	FUNCTION FC 833  : VOID
	TITLE =MAL1S033 Section control: LINE 1 SEC 33 KILN 2
	//COPYRIGHT:    (C) 2009 BY  BUHLER AG
	//                           CH-9240 UZWIL  SWITZERLAND
	//
	//PRODUCT:      WinCoS_BIW01_09
	//
	//TITLE:        LINE 1 SEC 33 KILN 2
	//                 Section control
	//
	//--------------------------------------------------------------------------------
	//
	//IDENT:        AUTHOR:             DEPT:                              DATE:
	//
	//P01_FC833.1.0 K.Renz              CSB41                              20.Okt.2009
	//              1st Release
	//
	//--------------------------------------------------------------------------------
	//
	//PURPOSE:
	//
	//REFERENCES : GCSOSMAN
	//
	//--------------------------------------------------------------------------------
	//
	//
	AUTHOR  : KR
	FAMILY  : USW
	VERSION : 9.9
	//0000 to 0999: Main Functions
	//              0 =Main Function Cylic
	//              1 =Main Function Coldstart/Newstart
	//              2 =Main Function Warm Start

	VAR_INPUT
	  InCode : INT ;
	END_VAR

	VAR_TEMP
	tmpStartNext : BOOL ;	//Condition to Start next element
	tmpFlagFault : BOOL ;	//Flag mechanical fault
	tmpEnableFeed : BOOL ;
	tmpStartScale : BOOL ;
	tmpStartLiqScale : BOOL ; //Enable to Start Lipquid Scale
	tmpSndBin: Int ;
	tmpRcvBin: Int ;
	tmpBool : BOOL ;
	tmpByte : BYTE ;
	tmpWord : WORD ;
	tmpDWord : DWORD ;
	tmpInt : INT ;
	tmpRET : INT ;
	tmpDInt : DINT ;
	tmpCyclusTime : DINT ;
	tmpWetSteep : BOOL ;
	END_VAR

	BEGIN

	NETWORK
	TITLE =
	//=================================================
	//=================================================
	//S T A R T   M A I N   F U N C T I O N
	//=================================================
	//=================================================
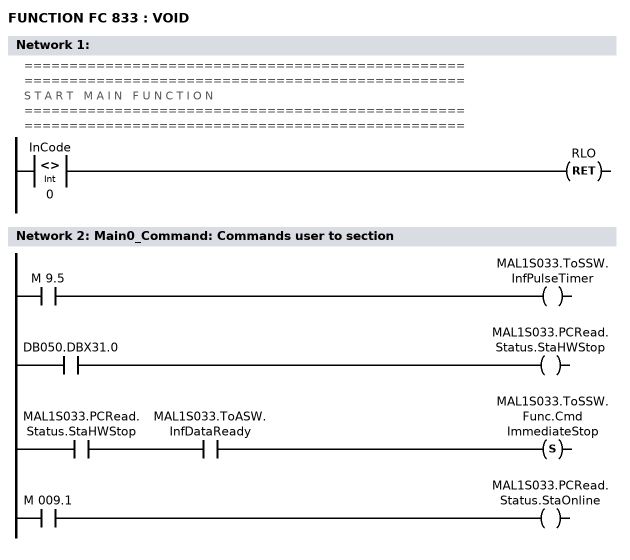
	      L InCode;
	      L 0;
	      <>I;
	      BEB;

	NETWORK
	TITLE =Main0_Command: Commands user to section
	      NOP   0;
	//-Tick 1 second---
		U     M 9.5;
		=     MAL1S033.ToSSW.InfPulseTimer;
	//-Hardware stop---
		U     DB050.DBX31.0 ;
		=     MAL1S033.PCRead.Status.StaHWStop;
		U   MAL1S033.PCRead.Status.StaHWStop;
		U   MAL1S033.ToASW.InfDataReady;
		S     MAL1S033.ToSSW.Func.CmdImmediateStop;
	//-Online---
		U     M 009.1 ;
		=     MAL1S033.PCRead.Status.StaOnline;
	NETWORK
	TITLE =ASW_UC: User commands to section
	NOP 0;
	//-Additional user commands---
	//-GP standard commands---
	      AUF   "MAL1S033" ;
	      L     L#0 ;                           // Enter the differenz of the target weight and prestop weight
	      T    "MAL1S033".VarTemp.InOutValue3;  // Prestop weight
	      CALL FC   120 (
	           InCode                   := 2001);// Section function: Standard section commands

	//-Condition CmdSequenzStop---
	      U     MAL1S033.ToSSW.Func.CmdSequenzStop;
	//      S     "MAL1S033".ToSSW.Func.CmdSequenzStop
	      R     MAL1S033.ToSSW.Func.CmdSequenzStop;
	//-Extended section commands---
	      AUF   "MAL1S033";
	      CALL "STD_LineSecStdSub" (
	           InCode                   := 2002);// Section function: Extended section commands
	//-Status from pulse commands---
	      CLR;
	      =     DB833.DBX  157.0;
	      =     DB833.DBX  157.1;
	      =     DB833.DBX  157.2;
	      =     DB833.DBX  157.3;
	      =     DB833.DBX  157.4;
	      =     DB833.DBX  157.5;
	      =     DB833.DBX  157.6;
	      =     DB833.DBX  157.7;
	//
	NETWORK
	TITLE =Main0_Dest: Destination
	NETWORK
	TITLE =Main0_Next: Ready for next batch

		ON    MAL1S033.ToASW.InfDataReady;
		=     MAL1S033.ToSSW.InfReadyForNewBatch;
	NETWORK
	TITLE =Main0_Control: Control section
	      NOP   0;
	//-Process commands from PCS---
		AUF   "MAL1S033" ;
		CALL FC    60 (// Methode O_Section
		CODE                     := 7);
	//-Process commands from user---
		AUF   "MAL1S033" ;
		CALL FC    60 (// Methode Control
		CODE                     := 0);
	//-Process section step---
		AUF   "MAL1S033" ;
		CALL FC    60 (// Methode Step_execute
		CODE                     := 2);
		AUF   "MAL1S033" ;
		CALL FC    60 (// Methode Step_transition
		CODE                     := 3);
	//-Process section state---
		AUF   "MAL1S033" ;
		CALL FC    60 (// Methode State
		CODE                     := 4);

	NETWORK
	TITLE =Main0_Init: Init
		UN    MAL1S033.ToASW.Transition.ToWait;
		UN    MAL1S033.ToASW.CmdNewBatch;
		SPB   in00;
	//-User initialization---
		AUF   "MAL1S033" ;
	//
	//-Section function: Init ---
		AUF   "MAL1S033" ;
	      CALL FC   120 (
	           InCode                   := 2003);// Section function: Init
	//
	//-Group interface---
	//
	//-Initialise bin objects---
	//
	//-Emptying job---
	      U    MAL1S033.JobAc.StaBatch.StaEmptyingBatch;
	      S     MAL1S033.PCRead.Status.StaLoaded;
	//
	//-Error Batch---
	//
	in00:	NOP   0;

	NETWORK
	TITLE =ASW_VB: Various functions before bin control
	      NOP   0;
	//
	//-Update staSameSndRcv in sender binlist---
	NETWORK
	TITLE =Main0_GrNRS: Not Relevant for started / Fault
		NOP 0;
	NETWORK
	TITLE =Main0_GrSelection: Group selection
	// List of the used objects in the section
	// ==========================
	// G022G       GENERAL ELEMENTS KILN 2
	// G261M       BELT CONVEYOR 7200 KILN
	// G262M       BELT CONVEYOR 7300 KILN
	// G263M       BELT CONVEYOR 7301 KILN
	// G264M       BELT CONVEYOR 7400 KILN
	// G291M       LIFTING DEVICE KILN 2
	// G292M       TRAVELLING DRIVE KILN 2
	// G293M       UNLOADING / LOADING SCREW KILN 2
	// G294M       DISCHARGE DOOR KILN 2
	// G295M       TEMPERATURE MES. KILN 2
	// G296M       AIR SHUT SLIDE KILN 2
	// G297M       FAN KILN 2
	// G298M       FRESH AIR LOUVER KILN 2
	// G299M       RECYCLING AIR FLAP KILN 2
	// G300M       EXHAUST AIR FLAP KILN 2
	// G301M       LOUVER HEATING GLASS TUBE HEAT EXCHANGER
	// G302M       HEATING KILN 2
	// G303M       LOUVER AIR HEATER KILN 2
	// G304M       WITHERING AIR KILN 2
	// G279M       HEATING KILN 1 + 2
	// G305M       CHAIN CONVEYOR 9002 KILN 2
	// G281M       ELEVATOR 9002 AFTER KILN
	// G282M       FLAP BOX 9008
	// G283M       CULM BATCH BIN 9005
	//
	      NOP   0;
//-Condition for preselection---
		U     MAL1S033.ToASW.InfDataReady;
		SPB   GS01;
//-Deselect groups ---
		CALL FB     9 , "GCS7_GrCtrlDBTmp" (// GrCtr.Methode Deselect
		     Code  := 3,
		     Sec   := "MAL1S033".Gr);
		SPA   GS02;
//-Select groups ---
	GS01:	NOP 0;
	//-Prepare for preselection ---
		CALL FB     9 , "GCS7_GrCtrlDBTmp" (// GrCtr.Methode Init Preselection
		     Code  := 1,
		     Sec   := "MAL1S033".Gr);
	//
	//
	//-Prestart used groups --
		U     M     50.0;
		=     M     50.0;

	//-Preselect used groups --
		U     M     50.0;
		=     M     50.0;
		S   MAL1S033.Gr.InPreselect[22];   //-->G022G GENERAL ELEMENTS KILN 2
		S   MAL1S033.Gr.InPreselect[261];   //-->G261M BELT CONVEYOR 7200 KILN
		S   MAL1S033.Gr.InPreselect[262];   //-->G262M BELT CONVEYOR 7300 KILN
		S   MAL1S033.Gr.InPreselect[263];   //-->G263M BELT CONVEYOR 7301 KILN
		S   MAL1S033.Gr.InPreselect[264];   //-->G264M BELT CONVEYOR 7400 KILN
		S   MAL1S033.Gr.InPreselect[291];   //-->G291M LIFTING DEVICE KILN 2
		S   MAL1S033.Gr.InPreselect[292];   //-->G292M TRAVELLING DRIVE KILN 2
		S   MAL1S033.Gr.InPreselect[293];   //-->G293M UNLOADING / LOADING SCREW KILN 2
		S   MAL1S033.Gr.InPreselect[294];   //-->G294M DISCHARGE DOOR KILN 2
		S   MAL1S033.Gr.InPreselect[295];   //-->G295M TEMPERATURE MES. KILN 2
		S   MAL1S033.Gr.InPreselect[296];   //-->G296M AIR SHUT SLIDE KILN 2
		S   MAL1S033.Gr.InPreselect[297];   //-->G297M FAN KILN 2
		S   MAL1S033.Gr.InPreselect[298];   //-->G298M FRESH AIR LOUVER KILN 2
		S   MAL1S033.Gr.InPreselect[299];   //-->G299M RECYCLING AIR FLAP KILN 2
		S   MAL1S033.Gr.InPreselect[300];   //-->G300M EXHAUST AIR FLAP KILN 2
		S   MAL1S033.Gr.InPreselect[301];   //-->G301M LOUVER HEATING GLASS TUBE HEAT EXCHANGER
		S   MAL1S033.Gr.InPreselect[302];   //-->G302M HEATING KILN 2
		S   MAL1S033.Gr.InPreselect[303];   //-->G303M LOUVER AIR HEATER KILN 2
		S   MAL1S033.Gr.InPreselect[304];   //-->G304M WITHERING AIR KILN 2
		S   MAL1S033.Gr.InPreselect[279];   //-->G279M HEATING KILN 1 + 2
		S   MAL1S033.Gr.InPreselect[305];   //-->G305M CHAIN CONVEYOR 9002 KILN 2
		S   MAL1S033.Gr.InPreselect[281];   //-->G281M ELEVATOR 9002 AFTER KILN
		S   MAL1S033.Gr.InPreselect[282];   //-->G282M FLAP BOX 9008
		S   MAL1S033.Gr.InPreselect[283];   //-->G283M CULM BATCH BIN 9005
	      L     1;
	      L     "MAL1S033Par".StepAct.StepNumber;
	      UW;
	      ==I;  // step wetsteep
	      =    "MAL1S033Par".Par.FlagGen.WetStep;

	//
	//-Set CmdNewJob ---
	     U     MAL1S033.Gr.InPreselect[261];
	     UN    #GCS7_GrCtrlDB.OutOccupied[261];
	     S       G261M.CmdNewJob;
	     U     MAL1S033.Gr.InPreselect[262];
	     UN    #GCS7_GrCtrlDB.OutOccupied[262];
	     S       G262M.CmdNewJob;
	     U     MAL1S033.Gr.InPreselect[263];
	     UN    #GCS7_GrCtrlDB.OutOccupied[263];
	     S       G263M.CmdNewJob;
	     U     MAL1S033.Gr.InPreselect[264];
	     UN    #GCS7_GrCtrlDB.OutOccupied[264];
	     S       G264M.CmdNewJob;
	     U     MAL1S033.Gr.InPreselect[291];
	     UN    #GCS7_GrCtrlDB.OutOccupied[291];
	     S       G291M.CmdNewJob;
	     U     MAL1S033.Gr.InPreselect[292];
	     UN    #GCS7_GrCtrlDB.OutOccupied[292];
	     S       G292M.CmdNewJob;
	     U     MAL1S033.Gr.InPreselect[293];
	     UN    #GCS7_GrCtrlDB.OutOccupied[293];
	     S       G293M.CmdNewJob;
	     U     MAL1S033.Gr.InPreselect[294];
	     UN    #GCS7_GrCtrlDB.OutOccupied[294];
	     S       G294M.CmdNewJob;
	     U     MAL1S033.Gr.InPreselect[295];
	     UN    #GCS7_GrCtrlDB.OutOccupied[295];
	     S       G295M.CmdNewJob;
	     U     MAL1S033.Gr.InPreselect[296];
	     UN    #GCS7_GrCtrlDB.OutOccupied[296];
	     S       G296M.CmdNewJob;
	     U     MAL1S033.Gr.InPreselect[297];
	     UN    #GCS7_GrCtrlDB.OutOccupied[297];
	     S       G297M.CmdNewJob;
	     U     MAL1S033.Gr.InPreselect[298];
	     UN    #GCS7_GrCtrlDB.OutOccupied[298];
	     S       G298M.CmdNewJob;
	     U     MAL1S033.Gr.InPreselect[299];
	     UN    #GCS7_GrCtrlDB.OutOccupied[299];
	     S       G299M.CmdNewJob;
	     U     MAL1S033.Gr.InPreselect[300];
	     UN    #GCS7_GrCtrlDB.OutOccupied[300];
	     S       G300M.CmdNewJob;
	     U     MAL1S033.Gr.InPreselect[301];
	     UN    #GCS7_GrCtrlDB.OutOccupied[301];
	     S       G301M.CmdNewJob;
	     U     MAL1S033.Gr.InPreselect[302];
	     UN    #GCS7_GrCtrlDB.OutOccupied[302];
	     S       G302M.CmdNewJob;
	     U     MAL1S033.Gr.InPreselect[303];
	     UN    #GCS7_GrCtrlDB.OutOccupied[303];
	     S       G303M.CmdNewJob;
	     U     MAL1S033.Gr.InPreselect[304];
	     UN    #GCS7_GrCtrlDB.OutOccupied[304];
	     S       G304M.CmdNewJob;
	     U     MAL1S033.Gr.InPreselect[279];
	     UN    #GCS7_GrCtrlDB.OutOccupied[279];
	     S       G279M.CmdNewJob;
	     U     MAL1S033.Gr.InPreselect[305];
	     UN    #GCS7_GrCtrlDB.OutOccupied[305];
	     S       G305M.CmdNewJob;
	     U     MAL1S033.Gr.InPreselect[281];
	     UN    #GCS7_GrCtrlDB.OutOccupied[281];
	     S       G281M.CmdNewJob;
	     U     MAL1S033.Gr.InPreselect[282];
	     UN    #GCS7_GrCtrlDB.OutOccupied[282];
	     S       G282M.CmdNewJob;
	     U     MAL1S033.Gr.InPreselect[283];
	     UN    #GCS7_GrCtrlDB.OutOccupied[283];
	     S       G283M.CmdNewJob;
	//
	//
	//-Test preselected groups ---
		CALL FB     9 , "GCS7_GrCtrlDBTmp" (// GrCtr.Methode Select
		     Code  := 2,
		     Sec   := "MAL1S033".Gr);
	//
	//-Way conflict if not available---
		CLR;
		S     MAL1S033.Gr.All.OutGrConflict;
	//
	//-Test occupied real and virtual groups---
	GS02:   NOP 0;
		U     MAL1S033.Gr.All.OutSelectionValid;
		UN    MAL1S033.Gr.All.OutGrIsLocked;
		=     MAL1S033.Gr.All.InOutASWSelectionOK;
	//
	//
	//----- Send data to selected groups =====
	GS3:	UN  MAL1S033.Gr.OutSelected[261]; //G261M
		SPB GS4;
		L     "MAL1".Para.ParLineNr;
		T     G261M.Gr.InLine;
	GS4:	UN  MAL1S033.Gr.OutSelected[262]; //G262M
		SPB GS5;
		L     "MAL1".Para.ParLineNr;
		T     G262M.Gr.InLine;
	GS5:	UN  MAL1S033.Gr.OutSelected[263]; //G263M
		SPB GS6;
		L     "MAL1".Para.ParLineNr;
		T     G263M.Gr.InLine;
	GS6:	UN  MAL1S033.Gr.OutSelected[264]; //G264M
		SPB GS7;
		L     "MAL1".Para.ParLineNr;
		T     G264M.Gr.InLine;
	GS7:	UN  MAL1S033.Gr.OutSelected[291]; //G291M
		SPB GS8;
		L     "MAL1".Para.ParLineNr;
		T     G291M.Gr.InLine;
	GS8:	UN  MAL1S033.Gr.OutSelected[292]; //G292M
		SPB GS9;
		L     "MAL1".Para.ParLineNr;
		T     G292M.Gr.InLine;
	GS9:	UN  MAL1S033.Gr.OutSelected[293]; //G293M
		SPB GS10;
		L     "MAL1".Para.ParLineNr;
		T     G293M.Gr.InLine;
	GS10:	UN  MAL1S033.Gr.OutSelected[294]; //G294M
		SPB GS11;
		L     "MAL1".Para.ParLineNr;
		T     G294M.Gr.InLine;
	GS11:	UN  MAL1S033.Gr.OutSelected[295]; //G295M
		SPB GS12;
		L     "MAL1".Para.ParLineNr;
		T     G295M.Gr.InLine;
	GS12:	UN  MAL1S033.Gr.OutSelected[296]; //G296M
		SPB GS13;
		L     "MAL1".Para.ParLineNr;
		T     G296M.Gr.InLine;
	GS13:	UN  MAL1S033.Gr.OutSelected[297]; //G297M
		SPB GS14;
		L     "MAL1".Para.ParLineNr;
		T     G297M.Gr.InLine;
	GS14:	UN  MAL1S033.Gr.OutSelected[298]; //G298M
		SPB GS15;
		L     "MAL1".Para.ParLineNr;
		T     G298M.Gr.InLine;
	GS15:	UN  MAL1S033.Gr.OutSelected[299]; //G299M
		SPB GS16;
		L     "MAL1".Para.ParLineNr;
		T     G299M.Gr.InLine;
	GS16:	UN  MAL1S033.Gr.OutSelected[300]; //G300M
		SPB GS17;
		L     "MAL1".Para.ParLineNr;
		T     G300M.Gr.InLine;
	GS17:	UN  MAL1S033.Gr.OutSelected[301]; //G301M
		SPB GS18;
		L     "MAL1".Para.ParLineNr;
		T     G301M.Gr.InLine;
	GS18:	UN  MAL1S033.Gr.OutSelected[302]; //G302M
		SPB GS19;
		L     "MAL1".Para.ParLineNr;
		T     G302M.Gr.InLine;
	GS19:	UN  MAL1S033.Gr.OutSelected[303]; //G303M
		SPB GS20;
		L     "MAL1".Para.ParLineNr;
		T     G303M.Gr.InLine;
	GS20:	UN  MAL1S033.Gr.OutSelected[304]; //G304M
		SPB GS21;
		L     "MAL1".Para.ParLineNr;
		T     G304M.Gr.InLine;
	GS21:	UN  MAL1S033.Gr.OutSelected[279]; //G279M
		SPB GS22;
		L     "MAL1".Para.ParLineNr;
		T     G279M.Gr.InLine;
	GS22:	UN  MAL1S033.Gr.OutSelected[305]; //G305M
		SPB GS23;
		L     "MAL1".Para.ParLineNr;
		T     G305M.Gr.InLine;
	GS23:	UN  MAL1S033.Gr.OutSelected[281]; //G281M
		SPB GS24;
		L     "MAL1".Para.ParLineNr;
		T     G281M.Gr.InLine;
	GS24:	UN  MAL1S033.Gr.OutSelected[282]; //G282M
		SPB GS25;
		L     "MAL1".Para.ParLineNr;
		T     G282M.Gr.InLine;
	GS25:	UN  MAL1S033.Gr.OutSelected[283]; //G283M
		SPB GS26;
		L     "MAL1".Para.ParLineNr;
		T     G283M.Gr.InLine;
	GS26:	NOP 0;
	NETWORK
	TITLE =Main0_GrCmd: CMD section to Groups

		NOP   0;
//-Way Adjust Time---
		O     MAL1S033.Gr.All.CmdNewSelection;
		O     MAL1S033.ToASW.CmdModify;
		S     MAL1S033.ToSSW.CmdNewWay;
		AUF   "MAL1S033" ;
		CALL FC    60 (// Methode Adjust Time
		CODE                     := 13);
//-Continue---
		U     MAL1S033.ToASW.Func.CmdStart;
		O     MAL1S033.ToASW.Func.CmdNextStep;
		S     MAL1S033.Gr.All.CmdContinue;
//-Fault reset---
		U     MAL1S033.ToASW.Func.CmdFaultReset;
		S     MAL1S033.Gr.All.CmdFaultReset;
//-Manual mode---
		U     MAL1S033.ToASW.Func.CmdAutomatic;
		S     MAL1S033.Gr.All.CmdManualOff;
		UN     MAL1S033.PCRead.Status.StaHand;
		S     MAL1S033.Gr.All.CmdManualOffRel;
//-Clear idling---
		U     MAL1S033.PCRead.Status.StaImmediateStopASW;
		S     MAL1S033.Gr.All.CmdClearIdling;
//-Start next---
		UN    MAL1S033.PCRead.Status.StaStep;
		O     MAL1S033.ToASW.Func.CmdNextStep;
		U(;
		L       MAL1S033.PCRead.OutWayAdjustTime;
		L     2;
		>I;
		O     MAL1S033.ToASW.InfWayAdjustTimeEnd;
		);
		UN    MAL1S033.Gr.All.CmdNewSelection;
		UN    MAL1S033.PCRead.Step.StWait;
		=     #tmpStartNext; //-->VarStartNext
//-Start next feed---
		U     MAL1S033.Gr.Wgr.OutStartedRel;
		ON    MAL1S033.ToASW.InfWayAdjustTimeEnd;
		UN    MAL1S033.PCRead.Status.StaFeedOffASW;
		UN    MAL1S033.PCRead.Status.StaImmediateStopASW;
		U     MAL1S033.Gr.Mgr.OutStartedRel;
		U     MAL1S033.PCRead.Step.StActive;
		=     MAL1S033.Gr.Feed.InEnable;
		=     #tmpEnableFeed;
		U     #tmpStartNext;
		U     MAL1S033.Gr.Wgr.OutStartedRel;
		U     MAL1S033.Gr.All.OutAutoStartOk;
		U     MAL1S033.PCRead.Status.StaAutostartSec;
		=     MAL1S033.Gr.Feed.CmdNext;
//-Start next machine group---
		UN    MAL1S033.PCRead.Status.StaImmediateStopASW;
		=     MAL1S033.Gr.Mgr.InEnable;
		U     #tmpStartNext;
		=     MAL1S033.Gr.Mgr.CmdNext;
//-Start next way group---
		UN    MAL1S033.PCRead.Status.StaImmediateStopASW;
		=     MAL1S033.Gr.Wgr.InEnable;
		UN    MAL1S033.PCRead.Status.StaStep;
		O     MAL1S033.ToASW.Func.CmdNextStep;
		=     MAL1S033.Gr.Wgr.CmdNext;
//-Start next general group---
		UN    MAL1S033.PCRead.Status.StaImmediateStopASW;
		=     MAL1S033.Gr.Ggr.InEnable;
		U     #tmpStartNext;
		=     MAL1S033.Gr.Ggr.CmdNext;
//-Update command state---
		CALL FB     9 , "GCS7_GrCtrlDBTmp" (// GrCtr.Methode UpdateCmdSt
		     Code  := 4,
		     Sec   := "MAL1S033".Gr);

	NETWORK
	TITLE =Main0_Status: Fault/Status

		NOP   0;
//- Autostart Section---
		UN    MAL1S033.ToASW.Func.CmdStart;
		O     MAL1S033.Gr.All.OutAutoStartOk;
		=     MAL1S033.TimeoutAutostart.EN;
		CALL FC18 (
		   IN                       := MAL1S033.TimeoutAutostart.EN,
		   PT                       := 10,
		   Q                        := MAL1S033.TimeoutAutostart.Q,
		ET                       := MAL1S033.TimeoutAutostart.ET);
		U     MAL1S033.TimeoutAutostart.Q;
		UN     MAL1S033.Gr.All.OutAutoStartOk;
		R     MAL1S033.PCRead.Status.StaAutostartSec;
		U     MAL1S033.ToASW.Func.CmdStart;
		ON    MAL1S033.ToASW.InfDataReady;
		S     MAL1S033.PCRead.Status.StaAutostartSec;
//-Stopped---
		UN    MAL1S033.Gr.Mgr.InEnable;
		U     MAL1S033.Gr.All.OutStoppedRel;
		O     MAL1S033.Gr.All.OutStoppedAll;
		UN    MAL1S033.PCRead.Status.StaStep;
		O;
		U     MAL1S033.Gr.Mgr.OutStoppedRel;
		U     MAL1S033.PCRead.Status.StaStep;
		=     MAL1S033.ToSSW.InfStopped;
//-Started---
		U     MAL1S033.Gr.Mgr.OutStartedRel;
		=     MAL1S033.ToSSW.InfStarted;
//-Feeding---
		U     MAL1S033.Gr.Feed.InEnable; //Section without Feed groups
		ON    MAL1S033.Gr.Feed.OutStoppedAll;
		U     MAL1S033.Gr.Feed.OutStartedRel;
		=     MAL1S033.ToSSW.InfFeeding;
//-Autostart---
		U     MAL1S033.Gr.All.OutAutostartOkAll;
		U     MAL1S033.PCRead.Status.StaAutostartSec;
		=     MAL1S033.PCRead.Status.StaAutostart;
//-DPFault---
		U     MAL1S033.Gr.All.OutDPFault;
		=     MAL1S033.PCRead.Status.StaDPFault;
		S       MAL1S033.ToSSW.Func.CmdFeedOff;
//-Startwarning---
		U     MAL1S033.Gr.All.OutStartWarning;
		=     MAL1S033.PCRead.Status.StaStartwarning;
//-Way conflict---
		U     MAL1S033.Gr.All.OutGrConflict;
		=     MAL1S033.PCRead.Fault.EsWayConflict;
//-Warning---
		U     MAL1S033.Gr.All.OutWarning;
		=     MAL1S033.PCRead.Fault.EsWarning;
//-Fault---
		U     MAL1S033.Gr.All.OutFaultRel;
		FP      MAL1S033.PCRead.Fault.EsMech;
		S       MAL1S033.ToSSW.Func.CmdFeedOff;
//-Sender empty---
		CLR;
		=     MAL1S033.PCRead.Fault.EsEmpty; //-->Sec.EsEmpty
//-Receiver full---
		CLR;
		=     MAL1S033.PCRead.Fault.EsFull;

	NETWORK
	TITLE =Main0_StatusASW: Status from ASW
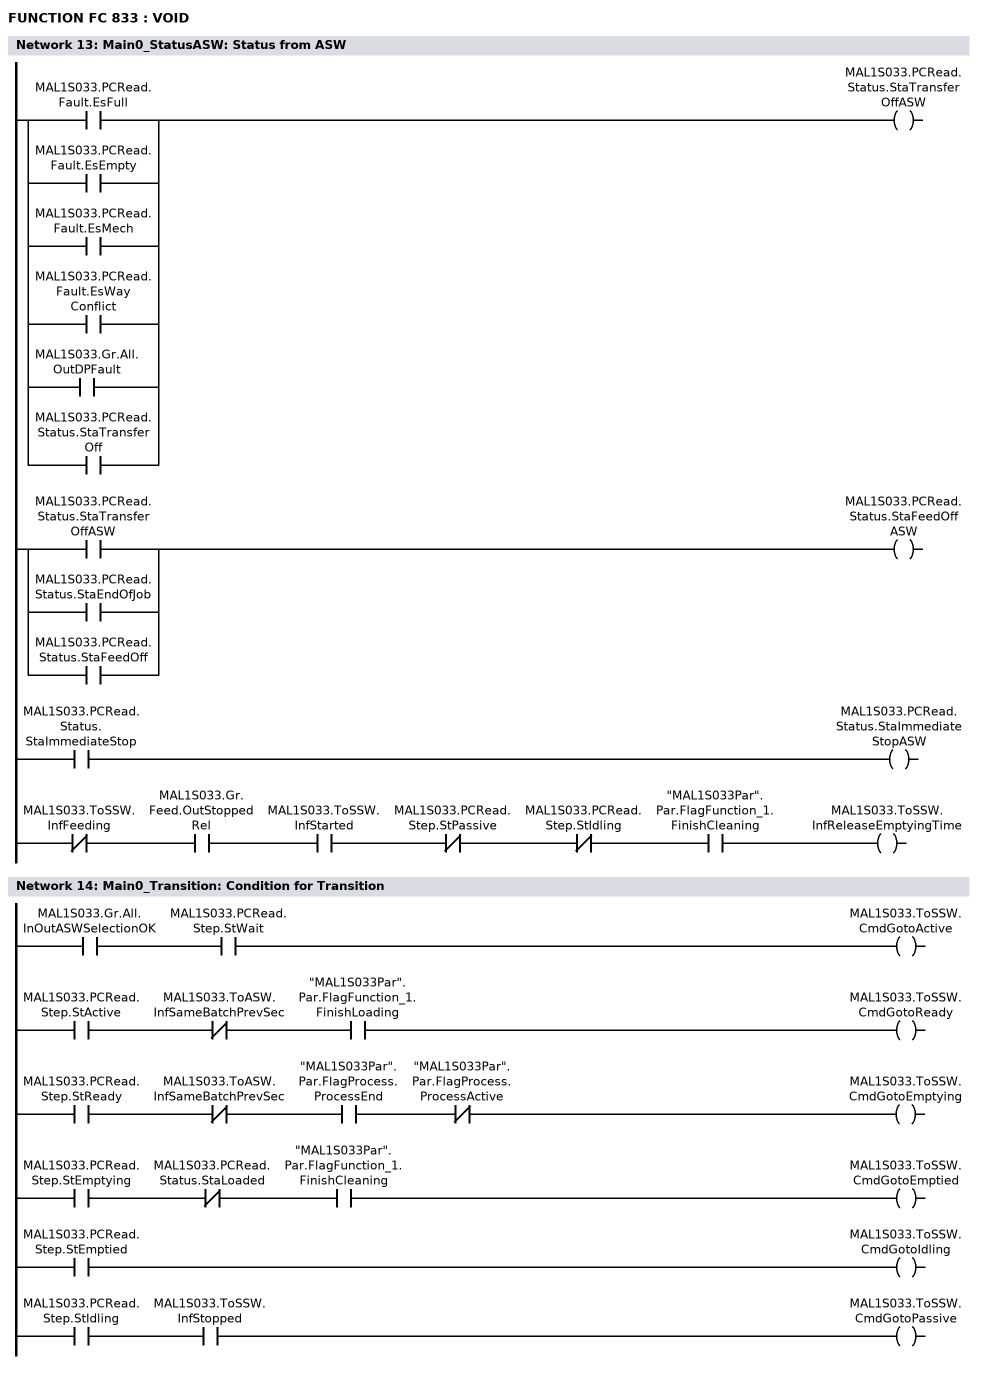
		NOP   0;
//-Transfer off with automatic restart---
		O     MAL1S033.PCRead.Fault.EsFull;
		O     MAL1S033.PCRead.Fault.EsEmpty;
		O     MAL1S033.PCRead.Fault.EsMech;
		O     MAL1S033.PCRead.Fault.EsWayConflict;
		O     MAL1S033.Gr.All.OutDPFault;
		O     MAL1S033.PCRead.Status.StaTransferOff;
		=     MAL1S033.PCRead.Status.StaTransferOffASW;
//-Feed off with automatic restart---
		U     MAL1S033.PCRead.Status.StaTransferOffASW;
		O     MAL1S033.PCRead.Status.StaEndOfJob; //
		O     MAL1S033.PCRead.Status.StaFeedOff;
		=     MAL1S033.PCRead.Status.StaFeedOffASW;
//-Immediate stop with automatic restart---
		U     MAL1S033.PCRead.Status.StaImmediateStop;
		=     MAL1S033.PCRead.Status.StaImmediateStopASW;
//-Emptying time---
	      UN   MAL1S033.ToSSW.InfFeeding;
	      U     MAL1S033.Gr.Feed.OutStoppedRel;
	      U     MAL1S033.ToSSW.InfStarted;
	      UN  MAL1S033.PCRead.Step.StPassive;
	      UN  MAL1S033.PCRead.Step.StIdling;
		U     "MAL1S033Par".Par.FlagFunction_1.FinishCleaning;
		=     MAL1S033.ToSSW.InfReleaseEmptyingTime;
	NETWORK
	TITLE =Main0_Transition: Condition for Transition

		NOP 0;
		NOP 0;
	//-Active---
		U   MAL1S033.Gr.All.InOutASWSelectionOK;
	        U    MAL1S033.PCRead.Step.StWait;
		=     MAL1S033.ToSSW.CmdGotoActive;
	//-Ready---
	        U    MAL1S033.PCRead.Step.StActive;
		UN   MAL1S033.ToASW.InfSameBatchPrevSec;
		U     "MAL1S033Par".Par.FlagFunction_1.FinishLoading;
		=     MAL1S033.ToSSW.CmdGotoReady;
	//-Emptying---
	        U    MAL1S033.PCRead.Step.StReady;
		UN   MAL1S033.ToASW.InfSameBatchPrevSec;
		U     "MAL1S033Par".Par.FlagProcess.ProcessEnd;
		UN    "MAL1S033Par".Par.FlagProcess.ProcessActive;
		=     MAL1S033.ToSSW.CmdGotoEmptying;
	//-Emptied---
	        U    MAL1S033.PCRead.Step.StEmptying;
		UN    MAL1S033.PCRead.Status.StaLoaded;
		U     "MAL1S033Par".Par.FlagFunction_1.FinishCleaning;
		=     MAL1S033.ToSSW.CmdGotoEmptied;
	//-Result section---
	//-Idling---
		U     MAL1S033.PCRead.Step.StEmptied;
		=     MAL1S033.ToSSW.CmdGotoIdling;
	//-Passive---
		U     MAL1S033.PCRead.Step.StIdling;
		U     MAL1S033.ToSSW.InfStopped;
		=     MAL1S033.ToSSW.CmdGotoPassive;
	NETWORK
	TITLE =Main0_Move: Move to next section
		NOP 0;
//-------------------------------------------
//-General Condition for move
//-------------------------------------------
		U   MAL1S033.PCRead.Step.StReady;
		SPBN  Move;
	//->Move batch to section MAL1S034
		AUF   "MAL1S033" ;
		CALL FC    60 (// Methode Move Data
		  CODE                     := 5);
		UN  MAL1S033.ToASW.CmdDataMoved;
		SPB Move;
	Move:	NOP 0;
	NETWORK
	TITLE =ASW_AH:Alarm horns
	      UN    MAL1S033.ToASW.Func.CmdHornOn;
	      SPB   AHJ1;
	      CALL "SYS_Horn_Code" (
	           FcCode                   := 1, //Set Alarm
	           ParObjectType            := 4000,
	           ParObjectNo              := 0,
	           ParHornCode              := 98);
	AHJ1: UN    MAL1S033.ToASW.Func.CmdHornOff;
	      SPB   AH00;
	      CALL "SYS_Horn_Code" (
	           FcCode                   := 2, //Reset Alarm
	           ParObjectType            := 4000,
	           ParObjectNo              := 0,
	           ParHornCode              := 10);
	      CALL "SYS_Horn_Code" (
	           FcCode                   := 2, //Reset Alarm
	           ParObjectType            := 4000,
	           ParObjectNo              := 0,
	           ParHornCode              := 11);
	      CALL "SYS_Horn_Code" (
	           FcCode                   := 2, //Reset Alarm
	           ParObjectType            := 4000,
	           ParObjectNo              := 0,
	           ParHornCode              := 12);
	AH00: NOP   0;
	NETWORK
	TITLE =ASW_FT: Feeding Time
		AUF   "MAL1S033" ;
	      CALL FC   120 (
	           InCode                 := 2004);// Section function: Feeding time

	NETWORK
	TITLE =ASW_OL: Override low level
	//
		AUF   "MAL1S033" ;
	//
	OL00: NOP   0;
	NETWORK
	TITLE =ASW_VA: VA Various functions after section control
	//
		AUF   "MAL1S033" ;
	// Copy bin number to section DB
	        L   MAL1S033.JobAc.BatchSndBin;
		L   MAL1S033.MAL1S001SND33.Ingr[1].Bin;
	        T   MAL1S033.JobAc.BatchSndBin;
		<>I;
		S   MAL1S033.ChangeBit.CBit1;
		//
	        L   MAL1S033.JobAc.BatchRcvBin;
		L   MAL1S033.MAL1S001RCV34.Ingr[1].Bin;
	        T   MAL1S033.JobAc.BatchRcvBin;
		<>I;
		S   MAL1S033.ChangeBit.CBit1;
		//
	        L   MAL1S033.JobAc.BatchRcvBin;
		L   MAL1S033.MAl1S034RCV36.Ingr[1].Bin;
	        T   MAL1S033.JobAc.BatchRcvBin;
		<>I;
		S   MAL1S033.ChangeBit.CBit1;
		//
	        L   MAL1S033.JobAc.BatchSndBin;
		L   MAL1S033.MAl1S034SND35.Ingr[1].Bin;
	        T   MAL1S033.JobAc.BatchSndBin;
		<>I;
		S   MAL1S033.ChangeBit.CBit1;
		//

	NETWORK
	TITLE =ASW_EJ End of job
	NOP 0;
	//
	//-Fluidlift monitoring---
	NETWORK
	TITLE =ASW_VE: VE New value event
	//
	//-Group interface---
	      U    MAL1S033.ToASW.CmdModify;
	      S     G261M.CmdNewValue;
	      S     G262M.CmdNewValue;
	      S     G263M.CmdNewValue;
	      S     G264M.CmdNewValue;
	      S     G291M.CmdNewValue;
	      S     G292M.CmdNewValue;
	      S     G293M.CmdNewValue;
	      S     G294M.CmdNewValue;
	      S     G295M.CmdNewValue;
	      S     G296M.CmdNewValue;
	      S     G297M.CmdNewValue;
	      S     G298M.CmdNewValue;
	      S     G299M.CmdNewValue;
	      S     G300M.CmdNewValue;
	      S     G301M.CmdNewValue;
	      S     G302M.CmdNewValue;
	      S     G303M.CmdNewValue;
	      S     G304M.CmdNewValue;
	      S     G279M.CmdNewValue;
	      S     G305M.CmdNewValue;
	      S     G281M.CmdNewValue;
	      S     G282M.CmdNewValue;
	      S     G283M.CmdNewValue;


	NETWORK
	TITLE =ASW_NV: New value data
	NETWORK
	TITLE =ASW_WJ: Weight job
	//
	      U     MAL1S033.PCRead.Step.StActive;
	      O     MAL1S033.PCRead.Step.StReady;
	      O     MAL1S033.PCRead.Step.StEmptying;
	      O     MAL1S033.PCRead.Step.StEmptied;
	      SPBN   WJ08;
	//
	      L     MAL1S033.JobNom.JobWeight; //Target/Actual registration if no scale
	      T     MAL1S033.JobAc.JobWeight;
	//
	WJ08: NOP 0;
	//--------------------------------------------
	//PW Prestop weight
	//--------------------------------------------
	WJ00: NOP   0;
	NETWORK
	TITLE =ASW_SC: Section status text and colour
	//
		AUF   "MAL1S033" ;
	      CALL FC   120 (
	           InCode                   := 2055);// Section function: WinCoS.SectionInfoCode
	//
	NETWORK
	TITLE =ASW_5010: Prepare Log-Data cyclic
	// Prepare Log-Data cyclic
	      U     "MAL1S033".ToASW.InfDataReady; // job in section
	      U     M      4.7; // scan 30sec
	      SPBN  N501;
	      AUF   "MAL1S033";
	      L     0;
	      T     #tmpInt;
	      CALL "SIEMENS_FILL" (
		   BVAL                     := #tmpInt,
		   RET_VAL                  := #tmpRet,
		   BLK                      := "SSA_LOG_Value_Queue".Input);
	// header
	//
	      L     B#16#1E; // type 30 = kilning
	      T     "SSA_LOG_Value_Queue".Input.Header.SecType; // type
	      L     B#16#1; // format 1 = cyclic
	      T     "SSA_LOG_Value_Queue".Input.Header.Format; // format
	      L     "MAL1S033".JobNom.JobNr;
	      T     "SSA_LOG_Value_Queue".Input.Para_0005;
	      L     "DB Prozesszeit".Sektion_33.Gesamtzeit_in_Minuten;
	      T     "SSA_LOG_Value_Queue".Input.Para_0007;
	      L     "MAL1S033Par".Par.ParIntMachine.ActualStep;
	      T     "SSA_LOG_Value_Queue".Input.Para_0008;
	      L     "MAL1S033Par".ActTimeStepProcess.SteptimeActMinOverall;
	      T     "SSA_LOG_Value_Queue".Input.Para_0009;
	//
	// values doubleword
	//=================================
	      L     G295M.A_3291_BTE07.OutValueUnits; // AIR TEMPERATURE ABOVE FLOOR
	      T     "SSA_LOG_Value_Queue".Input.Para_0015;
	//=================================
	      L     G295M.A_3291_BTE10.OutValueUnits; // AIR TEMPERATURE BEFORE BURNER 3
	      T     "SSA_LOG_Value_Queue".Input.Para_0017;
	//=================================
	      L     G295M.A_3291_BTE01.OutValueUnits; // AIR TEMPERATURE BELOW FLOOR
	      T     "SSA_LOG_Value_Queue".Input.Para_0019;
	//=================================
	//P4 setpoint from SCAD
	      L     "MAL1S033Par".StepAct.TemperaturBelowFloor; // setpoint from SCADA
	      T     "SSA_LOG_Value_Queue".Input.Para_0021;
	//=================================
	      L     G269M.A_3191_BTE11.OutValueUnits; // AIR TEMPERATURE AMBIENT AIR
	      T     "SSA_LOG_Value_Queue".Input.Para_0023;
	//=================================
	      L     G295M.A_3291_BTE05.OutValueUnits; // AIR TEMPERATURE DIFFUSOR FAN 1
	      T     "SSA_LOG_Value_Queue".Input.Para_0025;
	//=================================
	      L     G295M.A_3291_BTE08.OutValueUnits; // AIR TEMPERATURE AFTER BURNER 1
	      T     "SSA_LOG_Value_Queue".Input.Para_0027;
	//=================================
	      L     G269M.A_3191_BTE12.OutValueUnits; // AIR TEMPERATURE AFTER HEAT EXCHANGER FLAP
	      T     "SSA_LOG_Value_Queue".Input.Para_0029;
	//=================================
	      L     0; // act value airpressure after heatexchanger
	      T     "SSA_LOG_Value_Queue".Input.Para_0031;
	//=================================
	      L     0; // act value product temperature lowpoint
	      T     "SSA_LOG_Value_Queue".Input.Para_0033;
	//=================================
	      L     0; // act value product temperature middlepoint
	      T     "SSA_LOG_Value_Queue".Input.Para_0035;
	//=================================
	      L     0; // act value product temperature highpoint
	      T     "SSA_LOG_Value_Queue".Input.Para_0037;
	//=================================
	      L     0; // act value steam flowrate
	      T     "SSA_LOG_Value_Queue".Input.Para_0039;
	//=================================
	      L     0; // act value steam preasure inlet heatexchanger 1
	      T     "SSA_LOG_Value_Queue".Input.Para_0041;
	//=================================
	      L     0; // act value steam preasure inlet heatexchanger 2
	      T     "SSA_LOG_Value_Queue".Input.Para_0043;
	//=================================
	      L     0; // act value temperature steam inlet heatexchanger 1
	      T     "SSA_LOG_Value_Queue".Input.Para_0045;
	//=================================
	      L     0; // act value temperature steam inlet heatexchanger 2
	      T     "SSA_LOG_Value_Queue".Input.Para_0047;
	//=================================
	      L     0; // act position valve1 steam inlet heatexchanger 1
	      T     "SSA_LOG_Value_Queue".Input.Para_0049;
	//=================================
	      L     0; // act position valve2 steam inlet heatexchanger 1
	      T     "SSA_LOG_Value_Queue".Input.Para_0051;
	//=================================
	      L     0; // act position valve1 steam inlet heatexchanger 2
	      T     "SSA_LOG_Value_Queue".Input.Para_0053;
	//=================================
	      L     0; // act position valve2 steam inlet heatexchanger 2
	      T     "SSA_LOG_Value_Queue".Input.Para_0055;
	//=================================
	      L     0; // act value position exhaust air flap
	      T     "SSA_LOG_Value_Queue".Input.Para_0057;
	//=================================
	      L     0; // act value position recycling air flap
	      T     "SSA_LOG_Value_Queue".Input.Para_0059;
	//=================================
	      L     0; // act value position exhaust air flap to existing kiln
	      T     "SSA_LOG_Value_Queue".Input.Para_0061;
	//=================================
	      L     0; // act value position exhaust air flap
	      T     "SSA_LOG_Value_Queue".Input.Para_0063;
	//=================================
	      L     0; // act value position fresh air flap
	      T     "SSA_LOG_Value_Queue".Input.Para_0065;
	//=================================
	      L     0; // act value speed fan 1
	      T     "SSA_LOG_Value_Queue".Input.Para_0067;
	//=================================
	      L     0; // act value speed fan 2
	      T     "SSA_LOG_Value_Queue".Input.Para_0069;
	//=================================
	      L     0; // act value temperature bearing 1 fan 1
	      T     "SSA_LOG_Value_Queue".Input.Para_0071;
	//=================================
	      L     0; // act value temperature bearing 2 fan 1
	      T     "SSA_LOG_Value_Queue".Input.Para_0073;
	//=================================
	      L     0; // act value vibration bearing 1 fan 1
	      T     "SSA_LOG_Value_Queue".Input.Para_0075;
	//=================================
	      L     0; // act value vibration bearing 2 fan 1
	      T     "SSA_LOG_Value_Queue".Input.Para_0077;
	//=================================
	      L     0; // act value temperature bearing 1 fan 2
	      T     "SSA_LOG_Value_Queue".Input.Para_0079;
	//=================================
	      L     0; // act value temperature bearing 2 fan 2
	      T     "SSA_LOG_Value_Queue".Input.Para_0081;
	//=================================
	      L     0; // act value vibration bearing 1 fan 1
	      T     "SSA_LOG_Value_Queue".Input.Para_0083;
	//=================================
	      L     0; // act value vibration bearing 2 fan 1
	      T     "SSA_LOG_Value_Queue".Input.Para_0085;
	//=================================
	      L     0; // spare
	      T     "SSA_LOG_Value_Queue".Input.Para_0087;
	// values integer
	//
	      L     L#0; // spare
	      T     "SSA_LOG_Value_Queue".Input.Para_0089;
	      U     M      9.0; // spare
	      L   1;
	      SPB MP90;
	      L   0;
	MP90: T     "SSA_LOG_Value_Queue".Input.Para_0090;
	      U     M      9.0; // spare
	      L   1;
	      SPB MP91;
	      L   0;
	MP91: T     "SSA_LOG_Value_Queue".Input.Para_0091;
	      U     M      9.0; // spare
	      L   1;
	      SPB MP92;
	      L   0;
	MP92: T     "SSA_LOG_Value_Queue".Input.Para_0092; // spare
	      U     M      9.0; // spare
	      L   1;
	      SPB MP93;
	      L   0;
	MP93: T     "SSA_LOG_Value_Queue".Input.Para_0093; // spare
	      U     M      9.0; // cleaning on/off
	      L   1;
	      SPB MP94;
	      L   0;
	MP94: T     "SSA_LOG_Value_Queue".Input.Para_0094; // spare
	      U     M      9.0; // spare
	      L   1;
	      SPB MP95;
	      L   0;
	MP95: T     "SSA_LOG_Value_Queue".Input.Para_0095; // spare
	      U     M      9.0; // spare
	      L   1;
	      SPB MP96;
	      L   0;
	MP96: T     "SSA_LOG_Value_Queue".Input.Para_0096; // spare
	      U     "MAL1S033Par".Par.FlagProcess.TurningFloor; // turning floor 0/1
	      L   1;
	      SPB MP97;
	      L   0;
	MP97: T     "SSA_LOG_Value_Queue".Input.Para_0097;  //  turning floor 0/1
	      U     "MAL1S033Par".Par.FlagProcess.Cooling_Activ; // cooling down 0/1
	      L   1;
	      SPB MP98;
	      L   0;
	MP98: T     "SSA_LOG_Value_Queue".Input.Para_0098;  // cooling down 0/1
	      NOP   0;
	      NOP   0;
	// cont log-messages
	      L     "SSA_LOG_Value_Queue".Input.Para_0099; // message counter
	      L     1;
	      +I    ;
	      T     "SSA_LOG_Value_Queue".Input.Para_0099; // message counter

	// put timestamp into message
	      CALL "SIEMENS_BLKMOV" (
	           SRCBLK                   := "DB Prozesszeit".Arbeitsbereich.dt2,
	           RET_VAL                  := #tmpInt,
	           DSTBLK                   := "SSA_LOG_Value_Queue".Input.TimeStamp);
	//
	      CALL "SSA_MH_LogEntry_ActValue" (
	           DBNumber                 := 1005);
	N501: NOP   0;
	NETWORK
	TITLE =ASW_5030: Prepare Log-Data step values
	NOP 0;
	NETWORK
	TITLE =ASW_5060: Prepare Log-Data events
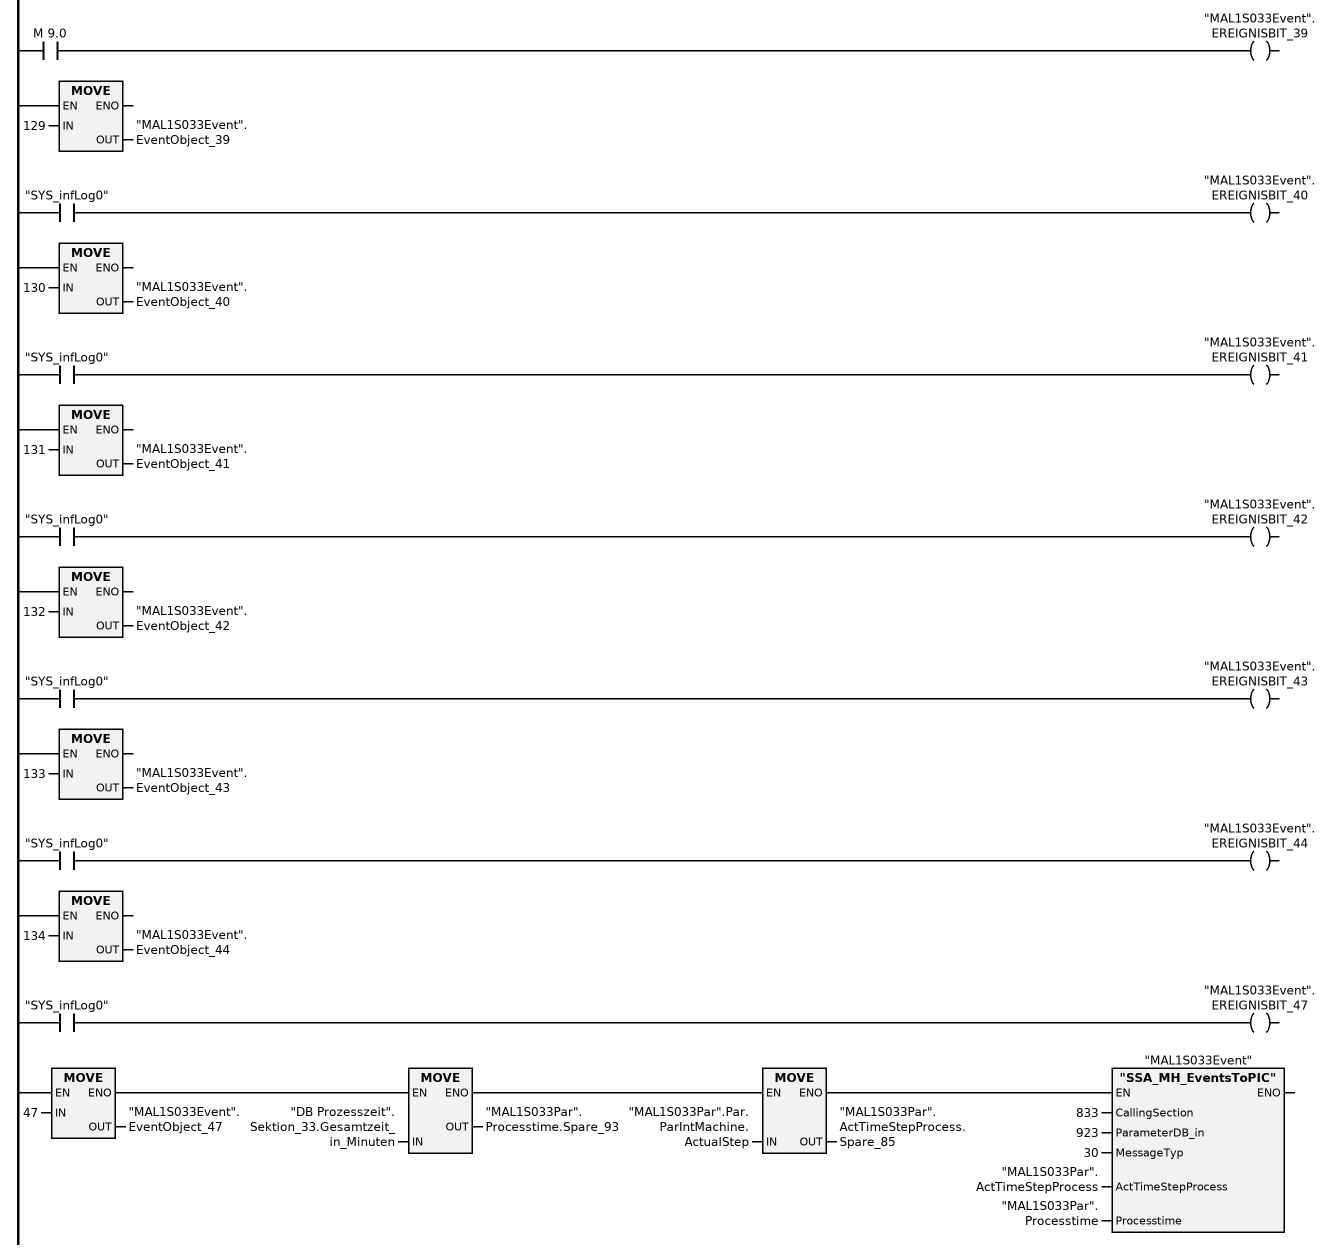
	NOP 0;
	// load events into event input

	// 1. event Process active
	      U     "MAL1S033Par".Par.FlagProcess.ProcessActive;
	      =     "MAL1S033Event".EREIGNISBIT_1;
	      L     1;
	      T     "MAL1S033Event".EventObject_1;
	// 2. event InfDataReady
	      U     "MAL1S033".ToASW.InfDataReady;
	      =     "MAL1S033Event".EREIGNISBIT_2;
	      L     2;
	      T     "MAL1S033Event".EventObject_2;
	// 11. event
	      U     "MAL1S033Par".Par.FlagFunction_1.StepLoading; // Step loading
	      =     "MAL1S033Event".EREIGNISBIT_11;
	      L     1001;
	      T     "MAL1S033Event".EventObject_11;
	// 12. event Loading Round 1
	      U     "MAL1S033Par".Par.FlagFunction_1.StepLoading;
	      U(    ;
	      L     G292M.A_3211_MXZ41MA.Ma.OutCntRound;
	      L     L#0;
	      ==D   ;
	      )     ;
	      =     "MAL1S033Event".EREIGNISBIT_12;
	      L     1003;
	      T     "MAL1S033Event".EventObject_12;
	// 13. event Loading Round 2
	      U     "MAL1S033Par".Par.FlagFunction_1.StepLoading;
	      U(    ;
	      L     G292M.A_3211_MXZ41MA.Ma.OutCntRound;
	      L     L#1;
	      ==D   ;
	      )     ;
	      =     "MAL1S033Event".EREIGNISBIT_13;
	      L     1004;
	      T     "MAL1S033Event".EventObject_13;
	// 14. event Loading Round 3
	      U     "MAL1S033Par".Par.FlagFunction_1.StepLoading;
	      U(    ;
	      L     G292M.A_3211_MXZ41MA.Ma.OutCntRound;
	      L     L#2;
	      ==D   ;
	      )     ;
	      =     "MAL1S033Event".EREIGNISBIT_14;
	      L     1005;
	      T     "MAL1S033Event".EventObject_14;
	// 15. event Loading Round 4
	      U     "MAL1S033Par".Par.FlagFunction_1.StepLoading;
	      U(    ;
	      L     G292M.A_3211_MXZ41MA.Ma.OutCntRound;
	      L     L#3;
	      ==D   ;
	      )     ;
	      =     "MAL1S033Event".EREIGNISBIT_15;
	      L     1006;
	      T     "MAL1S033Event".EventObject_15;
	// 16. event Loading Round 5
	      U     "MAL1S033Par".Par.FlagFunction_1.StepLoading;
	      U(    ;
	      L     G292M.A_3211_MXZ41MA.Ma.OutCntRound;
	      L     L#4;
	      ==D   ;
	      )     ;
	      =     "MAL1S033Event".EREIGNISBIT_16;
	      L     1007;
	      T     "MAL1S033Event".EventObject_16;
	// 17. event Loading Round 6
	      U     "MAL1S033Par".Par.FlagFunction_1.StepLoading;
	      U(    ;
	      L     G292M.A_3211_MXZ41MA.Ma.OutCntRound;
	      L     L#5;
	      ==D   ;
	      )     ;
	      =     "MAL1S033Event".EREIGNISBIT_17;
	      L     1008;
	      T     "MAL1S033Event".EventObject_17;
	// 18. event  Program withering/kilning
	      U     "MAL1S033Par".Par.FlagProcess.ProcessActive;
	      =     "MAL1S033Event".EREIGNISBIT_18;
	      L     1043;
	      T     "MAL1S033Event".EventObject_18;
	// 19. event ILO-Mode
	      U     "MAL1S033".SecAc.Sta1On.Inf08; // ILO-Mode Section
	      =     "MAL1S033Event".EREIGNISBIT_19;
	      L     1026;
	      T     "MAL1S033Event".EventObject_19;
	// 20. event Unloading
	      U     "MAL1S033Par".Par.FlagFunction_1.StepUnloading;
	      =     "MAL1S033Event".EREIGNISBIT_20;
	      L     1020;
	      T     "MAL1S033Event".EventObject_20;
	// 21. event Unloading Round 1
	      U     "MAL1S033Par".Par.FlagFunction_1.StepUnloading;
	      U(    ;
	      L     G292M.A_3211_MXZ41MA.Ma.OutCntRound;
	      L     L#0;
	      ==D   ;
	      )     ;
	      =     "MAL1S033Event".EREIGNISBIT_21;
	      L     1053;
	      T     "MAL1S033Event".EventObject_21;
	// 22. event Unloading Round 2
	      U     "MAL1S033Par".Par.FlagFunction_1.StepUnloading;
	      U(    ;
	      L     G292M.A_3211_MXZ41MA.Ma.OutCntRound;
	      L     L#1;
	      ==D   ;
	      )     ;
	      =     "MAL1S033Event".EREIGNISBIT_22;
	      L     1054;
	      T     "MAL1S033Event".EventObject_22;
	// 23. event Unloading Round 3
	      U     "MAL1S033Par".Par.FlagFunction_1.StepUnloading;
	      U(    ;
	      L     G292M.A_3211_MXZ41MA.Ma.OutCntRound;
	      L     L#2;
	      ==D   ;
	      )     ;
	      =     "MAL1S033Event".EREIGNISBIT_23;
	      L     1055;
	      T     "MAL1S033Event".EventObject_23;
	// 24. event
	      U     M      9.0;
	      =     "MAL1S033Event".EREIGNISBIT_24;
	      L     114;
	      T     "MAL1S033Event".EventObject_24;
	// 25. event Cleaning finished
	      U     "MAL1S033Par".Par.FlagFunction_1.FinishCleaning;
	      =     "MAL1S033Event".EREIGNISBIT_25;
	      L     1032;
	      T     "MAL1S033Event".EventObject_25;
	// 26. event  Cooling active
	      U     "MAL1S033Par".Par.FlagProcess.Cooling_Activ;
	      =     "MAL1S033Event".EREIGNISBIT_26;
	      L     1037;
	      T     "MAL1S033Event".EventObject_26;
	// 27. event  Process end
	      U     "MAL1S033Par".Par.FlagProcess.ProcessEnd;
	      =     "MAL1S033Event".EREIGNISBIT_27;
	      L     1038;
	      T     "MAL1S033Event".EventObject_27;
	// 28. event
	      U     M      9.0;
	      =     "MAL1S033Event".EREIGNISBIT_28;
	      L     118;
	      T     "MAL1S033Event".EventObject_28;
	// 29. event
	      U     M      9.0;
	      =     "MAL1S033Event".EREIGNISBIT_29;
	      L     119;
	      T     "MAL1S033Event".EventObject_29;
	// 30. event  steam regulator 1 on
	      U     M      9.0;
	      =     "MAL1S033Event".EREIGNISBIT_30;
	      L     1067;
	      T     "MAL1S033Event".EventObject_30;
	// 31. event  steam regulator 2 on
	      U     M      9.0;
	      =     "MAL1S033Event".EREIGNISBIT_31;
	      L     1068;
	      T     "MAL1S033Event".EventObject_31;
	// 32. event  steam regulator 3 on
	      U     M      9.0;
	      =     "MAL1S033Event".EREIGNISBIT_32;
	      L     1069;
	      T     "MAL1S033Event".EventObject_32;
	// 33. event  steam regulator 4 on
	      U     M      9.0;
	      =     "MAL1S033Event".EREIGNISBIT_33;
	      L     1070;
	      T     "MAL1S033Event".EventObject_33;
	// 34. event
	      U     M      9.0;
	      =     "MAL1S033Event".EREIGNISBIT_34;
	      L     124;
	      T     "MAL1S033Event".EventObject_34;
	// 35. event
	      U     M      9.0;
	      =     "MAL1S033Event".EREIGNISBIT_35;
	      L     125;
	      T     "MAL1S033Event".EventObject_35;
	// 36. event
	      U     M      9.0;
	      =     "MAL1S033Event".EREIGNISBIT_36;
	      L     126;
	      T     "MAL1S033Event".EventObject_36;
	// 37. event
	      U     M      9.0;
	      =     "MAL1S033Event".EREIGNISBIT_37;
	      L     127;
	      T     "MAL1S033Event".EventObject_37;
	// 38. event
	      U     M      9.0;
	      =     "MAL1S033Event".EREIGNISBIT_38;
	      L     128;
	      T     "MAL1S033Event".EventObject_38;
	// 39. event
	      U     M      9.0;
	      =     "MAL1S033Event".EREIGNISBIT_39;
	      L     129;
	      T     "MAL1S033Event".EventObject_39;
	// 40. event
	      U     "SYS_infLog0";
	      =     "MAL1S033Event".EREIGNISBIT_40;
	      L     130;
	      T     "MAL1S033Event".EventObject_40;
	//
	// 41. event
	      U     "SYS_infLog0";
	      =     "MAL1S033Event".EREIGNISBIT_41;
	      L     131;
	      T     "MAL1S033Event".EventObject_41;
	// 42. event
	      U     "SYS_infLog0";
	      =     "MAL1S033Event".EREIGNISBIT_42;
	      L     132;
	      T     "MAL1S033Event".EventObject_42;
	// 43. event
	      U     "SYS_infLog0";
	      =     "MAL1S033Event".EREIGNISBIT_43;
	      L     133;
	      T     "MAL1S033Event".EventObject_43;
	// 44. event
	      U     "SYS_infLog0";
	      =     "MAL1S033Event".EREIGNISBIT_44;
	      L     134;
	      T     "MAL1S033Event".EventObject_44;
	// only for test
	// 47. event
	      U     "SYS_infLog0";
	      =     "MAL1S033Event".EREIGNISBIT_47;
	      L     47;
	      T     "MAL1S033Event".EventObject_47;

	// copy data for event-logging
	      L     "DB Prozesszeit".Sektion_33.Gesamtzeit_in_Minuten;
	      T     "MAL1S033Par".Processtime.Spare_93;
	      L     "MAL1S033Par".Par.ParIntMachine.ActualStep;
	      T     "MAL1S033Par".ActTimeStepProcess.Spare_85;

	//
	      CALL "SSA_MH_EventsToPIC" , "MAL1S033Event" (
	           CallingSection           := 833,
	           ParameterDB_in           := 923,
	           MessageTyp               := 30,
	           ActTimeStepProcess       := "MAL1S033Par".ActTimeStepProcess,
	           Processtime              := "MAL1S033Par".Processtime);
	NETWORK
	TITLE =ASW_6000: Start process kilning
	      U     "MAL1S033".ToASW.InfDataReady;
	      U     "MAL1S033".PCRead.Step.StActive;
	      UN    "MAL1S033Par".Par.FlagProcess.ProcessActive;
	      U     "MAL1S033Par".Par.FlagFunction_1.FinishLoading;
	      SPBN  e605;
	      SET   ;
	      S     "MAL1S033Par".Par.FlagProcess.ProcessActive;
	      R     "MAL1S033Par".Par.FlagFunction_1.StepLoading;
	      S     "MAL1S033Par".Par.FlagMachine.ImpulsNullstellung;
	e605: NOP   0;
	//
	      U     "MAL1S033Par".Par.FlagProcess.ProcessActive;
	      U     "MAL1S033Par".Par.FlagFunction_1.FinishLoading;
	      U     "MAL1S033Par".Par.FlagFunction_1.StepUnloading; // Step Unloading
	      R     "MAL1S033Par".Par.FlagFunction_1.FinishLoading;
	//
	      U     "MAL1S033Par".Par.FlagProcess.ProcessActive;
	      FP    "MAL1S033Par".Par.FlagProcess.StartProzess_FP;
	      =     "MAL1S033Par".Par.FlagProcess.StartProzess_SCAN;
	E605: NOP   0;
	NETWORK
	TITLE =ASW_6010: Process Kilning Active
	      U     "MAL1S033".ToASW.InfDataReady;
	      SPB   NoCl;
	// Clear process time in buffer
	      L     0;
	      T     "MAL1S033Par".ActTimeStepProcess.SteptimeActHour;
	      T     "MAL1S033Par".ActTimeStepProcess.SteptimeActMin;
	      T     "MAL1S033Par".ActTimeStepProcess.SteptimeActMinOverall;
	      T     "MAL1S033Par".Processtime.Day;
	      T     "MAL1S033Par".Processtime.Hour;
	      T     "MAL1S033Par".Processtime.Min;
	      T     "MAL1S033Par".Processtime.ProcessTimeActive;
	      L     L#0; // clear actual step time
	      T     "MAL1S033Par".Par.ProcessValue.StepTimeAct; // in ms
	NoCl: NOP   0;
	// Clear process time in buffer end
	      U     "MAL1S033Par".Par.FlagProcess.ProcessActive;
	      SPBN  E606;
	//-Actual process time---
	      U     "MAL1S033Par".Par.FlagProcess.StartProzess_SCAN;
	      SPBN  actk;
	      L     1; // Start process first step
	      T     "MAL1S033Par".Par.ParIntMachine.ActualStep;
	      T     "MAL1S033Par".Par.ProcessValue.StepNrActCopy;
	      SPA   neSk;
	actk: NOP   0;
	// Prozesszeit
	      L     "DB Prozesszeit".Sektion_33.Tage;
	      INC   1; // malters do not accept day 0!!
	      T     "MAL1S033Par".Processtime.Day;
	      L     "DB Prozesszeit".Sektion_33.Stunden;
	      T     "MAL1S033Par".Processtime.Hour; // Processtime in h
	      L     "DB Prozesszeit".Sektion_33.Minuten;
	      T     "MAL1S033Par".Processtime.Min; // Processtime in min
	      U     "DB Prozesszeit".Sektion_33.Prozess_aktiv; // active bit section 2
	      L      1;
	      SPB    nTa;
	      L      0;
	nTa:  T     "MAL1S033Par".Processtime.ProcessTimeActive;
	// Test new step
	      L     "MAL1S033Par".Par.ParIntMachine.ActualStep;
	      L     "MAL1S033Par".Par.ProcessValue.StepNrActCopy;
	      ==I   ;
	      SPB   olSk;
	neSk: NOP   0;
	      L     "MAL1S033Par".Par.ParIntMachine.ActualStep;
	      T     "MAL1S033Par".Par.ProcessValue.StepNrActCopy;
	//
	      L     L#0; // clear actual step time
	      T     "MAL1S033Par".Par.ProcessValue.StepTimeAct; // in ms
	      L     0;
	      T     "MAL1S033Par".ActTimeStepProcess.SteptimeActMinOverall; // Steptime in min overall
	//
	      U(    ;
	      L     "MAL1S033Par".Par.ParIntMachine.ActualStep;
	      L     "MAL1S033Par".RecipeHeader.NumberOfSteps;
	      >I    ;
	      )     ;
	      SPB   Pedk; // last step is finished
	      SET   ;
	      S     "MAL1S033StepValues".StartStep; // start step for average calculating
	      SPA E606   ; // to secure, that new step-data are copied
	olSk: NOP   0;
	      L     "ASW_GraphicData".General.CycleTime[1].Actual;
	      T     #tmpCyclusTime;
	//
	      SPBN  NoTi; // count steptime only when fan running and sensor alive
	      L     "MAL1S033Par".Par.ProcessValue.StepTimeAct; // in ms
	      L     #tmpCyclusTime;
	      +D    ;
	      T     "MAL1S033Par".Par.ProcessValue.StepTimeAct; // in ms
	NoTi: NOP   0;
	      L     "MAL1S033Par".Par.ProcessValue.StepTimeAct; // in ms
	      L     L#86400000; // ms/d
	      MOD   ;
	      L     L#3600000; // ms/h
	      /D    ;
	      T     "MAL1S033Par".ActTimeStepProcess.SteptimeActHour; // Steptime in h
	//
	      L     "MAL1S033Par".Par.ProcessValue.StepTimeAct;
	      L     L#3600000; // ms/h
	      MOD   ;
	      L     L#60000; // ms/min
	      /D    ;
	      T     "MAL1S033Par".ActTimeStepProcess.SteptimeActMin; // Steptime in min
	//
	      L     "MAL1S033Par".Par.ProcessValue.StepTimeAct;
	      L     L#60000; // ms/min
	      /D    ;
	      T     "MAL1S033Par".ActTimeStepProcess.SteptimeActMinOverall; // Steptime in min overall
	//
	// Next Step
	//
	//   Switch over to next step under conditions:
	//   or Maximal steptime
	//   or Minimal steptime
	//           and
	//               or no setpoint delta temp
	//               or atual value delta temp is ge setpoint deltatemp
	//                   and sensor is ok
	//           and
	// /              or no setpoint max temp above floor
	//              or atual value max temp above floor is ge setpoint max temp above floor
	//                  and sensor is ok
	// 1 Kriterium
	      U(    ;
	      L     "MAL1S033Par".ActTimeStepProcess.SteptimeActMinOverall; // Steptime in min overall
	      L     "MAL1S033Par".StepAct.StepTime_Max; // Target steptime actual step
	      >=I   ;
	      )     ;
	      O(    ;
	// 2 Kriterium
	      O(    ;
	      U(;
	      L     "MAL1S033Par".StepAct.DeltaTempSwitchpointStep;
	      L     0;
	      >=D    ;
	      )      ;
	// condition, if analogue input is not damaaged   //
	      U(    ;
	      -D    ; // delta temp actual
	      L     L#10;
	      /D    ;
	      L     "MAL1S033Par".StepAct.DeltaTempSwitchpointStep;
	      <D    ;
	      )     ;
	      )     ;
	// 3 Kriterium
	      O(    ;
	      U(    ;
	      L     "MAL1S033Par".StepAct.MaxTempAboveFloorStep;
	      L     L#0; // 0,0°C is illegally switchpoint for max. temperature
	      >D   ;
	      )     ;
	// condition, if analogue input is not damaaged   // MW R2.1
	      U(    ;
	      L     L#10;
	      /D    ;
	      L     "MAL1S033Par".StepAct.MaxTempAboveFloorStep;
	      >=D   ;
	      )     ;
	      )     ;
	// 4 Kriterium
	// and min. time
	      U(    ;
	      L     "MAL1S033Par".ActTimeStepProcess.SteptimeActMinOverall; // Steptime in min overall
	      L     "MAL1S033Par".StepAct.StepTime_Min; // Target steptime actual step
	      >=I   ;
	      )     ;
	      )     ;
	// and not cooling                                // UK 22.01.07
	      UN    "MAL1S033Par".Par.FlagProcess.Cooling_Activ;
	// 5 Kriterium
	      O(    ;
	      U     "MAL1S033Par".Par.FlagProcess.Cooling_Activ;
	      U(    ;
	      L     L#10;
	      /D    ;
	      L     "MAL1S033Par".StepAct.TemperaturAboveFloor;
	      <=D   ;
	      )     ;
	      O(    ;
	      L     "MAL1S033Par".Par.ParIntMachine.ActualStep;
	      L     27; // max. 26 Schritte
	      >=I   ;
	      )     ;
	      )     ;
	// and min. time
	      U(    ;
	      L     "MAL1S033Par".ActTimeStepProcess.SteptimeActMinOverall; // Steptime in min overall
	      L     "MAL1S033Par".StepAct.StepTime_Min; // Target steptime actual step
	      >=I   ;
	      )     ;
	      SPBN  E606;
	// send average step data to PIC
	      SET   ;
	      S     "MAL1S033StepValues".SendData; // send average step data to PIC
	// Next step
	      L     "MAL1S033Par".Par.ParIntMachine.ActualStep;
	      L     "MAL1S033Par".RecipeHeader.NumberOfSteps;
	      >I    ;
	      SPB   Pedk; // Last step is finished
	//
	      L     "MAL1S033Par".Par.ParIntMachine.ActualStep;
	      L     1;
	      +I    ;
	      T     "MAL1S033Par".Par.ParIntMachine.ActualStep;
	      L     0;
	      T     "MAL1S033Par".ActTimeStepProcess.SteptimeActMinOverall; // Steptime in min Overall
	      SPA   E606;
	Pedk: NOP   0; // Process has finished
	      SET   ;
	      R     "MAL1S033Par".Par.FlagProcess.ProcessActive;
	      R     "MAL1S033Par".Par.FlagProcess.Cooling_Activ;
	      S     "MAL1S033Par".Par.FlagProcess.ProcessEnd;
	//
	      L     0; // clear step number
	      T     "MAL1S033Par".Par.ParIntMachine.ActualStep;
	E606: NOP   0;
	NETWORK
	TITLE =ASW_6020: Copy recipe-data in Parameter DB
	//
	// Clear content recipe in buffer
	      L     0;
	      T     #tmpInt;
	      CALL "SIEMENS_FILL" (
		   BVAL                     := #tmpInt,
		   RET_VAL                  := #tmpRet,
		   BLK                      := "MAL1S033Par".RecipeHeader);
	//
	      U     "MAL1S033Par".Par.FlagFunction_1.StepLoading;
	      O(    ;
	      U     "MAL1S033Par".Par.FlagFunction_1.StepUnloading;
	      UN    "MAL1S033Par".Par.FlagProcess.ProcessActive;
	      )     ;
	      SPBN  No10;
	// Copy step loading,unloading,cleaning to parameterDB
	      CALL "SIEMENS_BLKMOV" (
		   SRCBLK                   := "MAL1S033".SecNom.Kiln2.RecipeHeader.Loading,
		   RET_VAL                  := "MAL1S033Par".Par.Error.Value,
		   DSTBLK                   := "MAL1S033Par".RecipeHeader.Loading);
	      CALL "SIEMENS_BLKMOV" (
		   SRCBLK                   := "MAL1S033".SecNom.Kiln2.RecipeHeader.Unloading,
		   RET_VAL                  := "MAL1S033Par".Par.Error.Value,
		   DSTBLK                   := "MAL1S033Par".RecipeHeader.Unloading);
	      CALL "SIEMENS_BLKMOV" (
		   SRCBLK                   := "MAL1S033".SecNom.Kiln2.RecipeHeader.Cleaning,
		   RET_VAL                  := "MAL1S033Par".Par.Error.Value,
		   DSTBLK                   := "MAL1S033Par".RecipeHeader.Cleaning);
	      SPA   E607;
	No10: NOP   0;
	      U     "MAL1S033Par".Par.FlagProcess.ProcessActive;
	      SPBN  E607;
	// Copy common parameter
	      CALL "SIEMENS_BLKMOV" (
		   SRCBLK                   := "MAL1S033".SecNom.Kiln2.RecipeHeader,
		   RET_VAL                  := "MAL1S033Par".Par.Error.Value,
		   DSTBLK                   := "MAL1S033Par".RecipeHeader);
	//
	// Copy step parameter
	      U(    ;
	      L     "MAL1S033Par".Par.ParIntMachine.ActualStep;
	      L     1;
	      <I    ;
	      )     ;
	      O(    ;
	      L     "MAL1S033Par".Par.ParIntMachine.ActualStep;
	      L     "MAL1S033Par".RecipeHeader.NumberOfSteps;
	      >I    ;
	      )     ;
	      SPB   E607; // error wrong step number
	      CALL "SYS_Copy_Array_Element" (
		   Source                   := "MAL1S033".SecNom.Kiln2.Step,
		   Destination              := "MAL1S033Par".StepAct,
		   Index                    := "MAL1S033Par".Par.ParIntMachine.ActualStep,
		   Fault                    := "MAL1S033Par".Par.Error.Bit);
	E607: NOP   0;
	NETWORK
	TITLE =ASW_6080: Active step kilning
	//
	      U     "MAL1S033Par".Par.FlagProcess.ProcessActive;
	      SPBN  E608;
	// copy stepnr for visu
	      L     "MAL1S033Par".Par.ParIntMachine.ActualStep;
	      T     "MAL1S033Par".Par.ParIntProcess.ActualStep;
	// basic speed  fans
	      L     "MAL1S033Par".StepAct.SpeedVentilatorBasic;
	      T     "MAL1S033Par".Par.ParIntProcess.SpeedVentilatorBasic;
	// basic position waste air flaps
	      L     "MAL1S033Par".StepAct.PosExhaustAirFlapBasic; // setpoint from recipe
	      L     10; // convert to 0.1%
	      *I    ;
	      T     "MAL1S033Par".Par.ParIntProcess.PosExhaustAirFlapBasic;
		// emergency kiln heating
	// fan 1
	      U(    ;
	      L      2#1;
	      L     "MAL1S033Par".RecipeHeader.DeselectVentilator; // emergency regime without fan 1
	      ==I;
	      );
	      L   0; //temperature in diffusor fan 1
	      SPBN  c1R1;
	      L   0; //temerature below floor1
	      L   0; //temperature in diffusor fan 2
	      <D    ;
	      SPBN  c1R1;
	      TAK   ;
	c1R1: T     "MAL1S033Par".Par.ParIntProcess.ActValueTemperature_R1;
	// fan 2
	      U(    ;
	      L      2#10;
	      L     "MAL1S033Par".RecipeHeader.DeselectVentilator; // emergency regime without fan 2
	      ==I;
	      );
	      L   0; //temperature in diffusor fan 2
	      SPBN  c1R2;
	      L   0; //temerature below floor1
	      L   0; //temperature in diffusor fan 1
	      <D    ;
	      SPBN  c1R2;
	      TAK   ;
	c1R2: T     "MAL1S033Par".Par.ParIntProcess.ActValueTemperature_R2;
	// cooling down
	      L     "MAL1S033Par".StepAct.CoolingDown;
	      L     1;
	      ==I;
	      S     "MAL1S033Par".Par.FlagProcess.Cooling_Activ;
	E608: NOP   0;
	NETWORK
	TITLE =ASW_6090: calculate heat quantity active kilning
	      L     L#0;
	      U     "MAL1S033Par".Par.FlagProcess.ProcessActive;
	      SPBN  n609; // no addition
	      SET   ;
	      S     "MAL1S033Par".Par.FlagProcess.Inf21; // add heat quantity
	      U     M      4.5; // scan 1sec
	      SPBN  E609;
	      L     "MAL1S033Par".Par.ProcessValue_Real.Value05; // heat quantity in kW
	      +R    ;
	      T     "MAL1S033Par".Par.ProcessValue_Real.Value05;
	      SPA   E609;
	n609: NOP   0;
	      U     "MAL1S033Par".Par.FlagProcess.Inf21; // add heat quantity
	      SPBN  E609;
	      R     "MAL1S033Par".Par.FlagProcess.Inf21; // add heat quantity
	      L     "MAL1S033Par".Par.ProcessValue_Real.Value05;
	      L     3.600000e+003;
	      /R    ; // from kWs to kWh
	      L     1.000000e+003;
	      /R    ; // from kWh to MWh
	      RND   ;
	      T     "MAL1S033Par".Par.ProcessValue_Real.Value06; // result to batch potokoll
	      L     0.000000e+000; // clear calculator
	      T     "MAL1S033Par".Par.ProcessValue_Real.Value05;
	E609: NOP   0;
	NETWORK
	TITLE =ASW_7000: Step loading kilning
	//
	      U     "MAL1S033".ToASW.InfDataReady;
	      U     "MAL1S033".PCRead.Step.StWait;
	      U     "MAL1S033".PCWrite.ExtFuncOn.StartLoading; // PIC command "start loading"
	      S     "MAL1S033Par".Par.FlagFunction_1.StepLoading; // Step loading
	      U     "MAL1S033".PCWrite.ExtFuncOn.StartLoading; // PIC command "start loading"
	      R     "MAL1S033".PCWrite.ExtFuncOn.StartLoading; // PIC command "start loading"
	//
	      U     "MAL1S033".ToASW.InfDataReady;
	      U     "MAL1S033".PCRead.Step.StActive;
	      U     "MAL1S033Par".Par.FlagFunction_1.StepLoading; // Step loading
	      SPB   e71;
	      R     "MAL1S033Par".Par.Switches1.StaOn00; // LiftingPositionRound_1
	      R     "MAL1S033Par".Par.Switches1.StaOn01; // LiftingPositionRound_2
	      R     "MAL1S033Par".Par.Switches1.StaOn02; // LiftingPositionRound_3
	      R     "MAL1S033Par".Par.Switches1.StaOn03; // LiftingPositionRound_4
	      R     "MAL1S033Par".Par.Switches1.StaOn04; // LiftingPositionRound_5
	      R     "MAL1S033Par".Par.Switches1.StaOn05; // LiftingPositionRound_6
	e71:  NOP   0;
	      U     "MAL1S033".ToASW.InfDataReady;
	      U     "MAL1S033".PCRead.Step.StActive;
	      U     "MAL1S033Par".Par.FlagFunction_1.StepLoading; // Step loading
	      SPBN  E700;
	      L     "MAL1S033Par".RecipeHeader.Loading.LiftingPositionRound_3;
	      L     20; // 20°
	      -I    ;
	      T     "MAL1S033Par".Par.ParIntMachine.LiftingPositionRound_4;
	      L     "MAL1S033Par".RecipeHeader.Loading.LoadingLevelRound_3;
	      L     "MAL1S033Par".RecipeHeader.Loading.OffsetLevelNextRound;
	      +I    ;
	      T     "MAL1S033Par".Par.ParIntMachine.LoadingLevelRound_4;
	//
	      L     "MAL1S033Par".Par.ParIntMachine.LiftingPositionRound_4;
	      L     20; // 20°
	      -I    ;
	      T     "MAL1S033Par".Par.ParIntMachine.LiftingPositionRound_5;
	      L     "MAL1S033Par".Par.ParIntMachine.LoadingLevelRound_4;
	      L     "MAL1S033Par".RecipeHeader.Loading.OffsetLevelNextRound;
	      +I    ;
	      T     "MAL1S033Par".Par.ParIntMachine.LoadingLevelRound_5;
	//
	      L     "MAL1S033Par".Par.ParIntMachine.LiftingPositionRound_5;
	      L     20; // 20°
	      -I    ;
	      T     "MAL1S033Par".Par.ParIntMachine.LiftingPositionRound_6;
	      L     "MAL1S033Par".Par.ParIntMachine.LoadingLevelRound_5;
	      L     "MAL1S033Par".RecipeHeader.Loading.OffsetLevelNextRound;
	      +I    ;
	      T     "MAL1S033Par".Par.ParIntMachine.LoadingLevelRound_6;
	//
	      L     3600;
	      L     G292M.A_3211_MXZ41MA.Ma.Par.ParTolPosition;
	      -I    ;
	      L     G292M.A_3211_MXZ41MA.Ma.OutPositionAngle;
	      <=I   ;
	      SPB   E700;
	//
	      L     G292M.A_3211_MXZ41MA.Ma.OutPositionAngle;
	      L     0;
	      <=I   ;
	      SPB   E700;
	//
	      L     G292M.A_3211_MXZ41MA.Ma.OutPositionAngle;
	      L     10;
	      /I    ;
	      T     "MAL1S033Par".Par.MachineValue.ISTWERT_FAHRANTRIEB_POSI;
	//
	      U     "MAL1S033Par".Par.FlagFunction_1.StepLoading; // Step loading
	      FP    "MAL1S033Par".Par.Switches1.StaOn08;
	      =     "MAL1S033Par".Par.Switches1.StaOn09; // scan start loading
	      U     "MAL1S033Par".Par.Switches1.StaOn09; // scan start loading
	      SPBN  e72;
	      R     "MAL1S033Par".Par.Switches1.StaOn00; // LiftingPositionRound_1
	      R     "MAL1S033Par".Par.Switches1.StaOn01; // LiftingPositionRound_2
	      R     "MAL1S033Par".Par.Switches1.StaOn02; // LiftingPositionRound_3
	      R     "MAL1S033Par".Par.Switches1.StaOn03; // LiftingPositionRound_4
	      R     "MAL1S033Par".Par.Switches1.StaOn04; // LiftingPositionRound_5
	      R     "MAL1S033Par".Par.Switches1.StaOn05; // LiftingPositionRound_6
	//
	e72:  NOP   0;
	//
	      U(    ;
	      L     G292M.A_3211_MXZ41MA.Ma.OutCntRound;
	      L     L#0;
	      ==D   ;
	      )     ;
	      U(    ;
	      L     "MAL1S033Par".Par.MachineValue.ISTWERT_FAHRANTRIEB_POSI;
	      L     "MAL1S033Par".RecipeHeader.Loading.LiftingPositionRound_1;
	      <I    ;
	      )     ;
	      S     "MAL1S033Par".Par.Switches1.StaOn00; // LiftingPositionRound_1
	//
	      U(    ;
	      L     G292M.A_3211_MXZ41MA.Ma.OutCntRound;
	      L     L#0;
	      ==D   ;
	      )     ;
	      U(    ;
	      L     "MAL1S033Par".Par.MachineValue.ISTWERT_FAHRANTRIEB_POSI;
	      L     "MAL1S033Par".RecipeHeader.Loading.LiftingPositionRound_1;
	      >=I   ;
	      )     ;
	      S     "MAL1S033Par".Par.Switches1.StaOn01; // LiftingPositionRound_2
	//
	      U     "MAL1S033Par".Par.Switches1.StaOn01; // LiftingPositionRound_2
	      R     "MAL1S033Par".Par.Switches1.StaOn00; // LiftingPositionRound_1
	//
	      U(    ;
	      L     G292M.A_3211_MXZ41MA.Ma.OutCntRound;
	      L     L#1;
	      ==D   ;
	      )     ;
	      U(    ;
	      L     "MAL1S033Par".Par.MachineValue.ISTWERT_FAHRANTRIEB_POSI;
	      L     "MAL1S033Par".RecipeHeader.Loading.LiftingPositionRound_2;
	      >=I   ;
	      )     ;
	      S     "MAL1S033Par".Par.Switches1.StaOn02; // LiftingPositionRound_3
	//
	      U     "MAL1S033Par".Par.Switches1.StaOn02; // LiftingPositionRound_3
	      R     "MAL1S033Par".Par.Switches1.StaOn01; // LiftingPositionRound_2
	      R     "MAL1S033Par".Par.Switches1.StaOn00; // LiftingPositionRound_1
	//
	      U(    ;
	      L     G292M.A_3211_MXZ41MA.Ma.OutCntRound;
	      L     L#2;
	      ==D   ;
	      )     ;
	      U(    ;
	      L     "MAL1S033Par".Par.MachineValue.ISTWERT_FAHRANTRIEB_POSI;
	      L     "MAL1S033Par".RecipeHeader.Loading.LiftingPositionRound_3;
	      >=I   ;
	      )     ;
	      S     "MAL1S033Par".Par.Switches1.StaOn03; // LiftingPositionRound_4
	//
	      U     "MAL1S033Par".Par.Switches1.StaOn03; // LiftingPositionRound_4
	      R     "MAL1S033Par".Par.Switches1.StaOn02; // LiftingPositionRound_3
	      R     "MAL1S033Par".Par.Switches1.StaOn01; // LiftingPositionRound_2
	      R     "MAL1S033Par".Par.Switches1.StaOn00; // LiftingPositionRound_1
	      U(    ;
	      L     G292M.A_3211_MXZ41MA.Ma.OutCntRound;
	      L     L#3;
	      ==D   ;
	      )     ;
	      U(    ;
	      L     "MAL1S033Par".Par.MachineValue.ISTWERT_FAHRANTRIEB_POSI;
	      L     "MAL1S033Par".Par.ParIntMachine.LiftingPositionRound_4;
	      >=I   ;
	      )     ;
	      S     "MAL1S033Par".Par.Switches1.StaOn04; // LiftingPositionRound_5
	//
	      U     "MAL1S033Par".Par.Switches1.StaOn04; // LiftingPositionRound_5
	      R     "MAL1S033Par".Par.Switches1.StaOn03; // LiftingPositionRound_4
	      R     "MAL1S033Par".Par.Switches1.StaOn02; // LiftingPositionRound_3
	      R     "MAL1S033Par".Par.Switches1.StaOn01; // LiftingPositionRound_2
	      R     "MAL1S033Par".Par.Switches1.StaOn00; // LiftingPositionRound_1
	      U(    ;
	      L     G292M.A_3211_MXZ41MA.Ma.OutCntRound;
	      L     L#4;
	      ==D   ;
	      )     ;
	      U(    ;
	      L     "MAL1S033Par".Par.MachineValue.ISTWERT_FAHRANTRIEB_POSI;
	      L     "MAL1S033Par".Par.ParIntMachine.LiftingPositionRound_5;
	      >=I   ;
	      )     ;
	      S     "MAL1S033Par".Par.Switches1.StaOn05; // LiftingPositionRound_6
	//
	      U     "MAL1S033Par".Par.Switches1.StaOn05; // LiftingPositionRound_6
	      R     "MAL1S033Par".Par.Switches1.StaOn04; // LiftingPositionRound_5
	      R     "MAL1S033Par".Par.Switches1.StaOn03; // LiftingPositionRound_4
	      R     "MAL1S033Par".Par.Switches1.StaOn02; // LiftingPositionRound_3
	      R     "MAL1S033Par".Par.Switches1.StaOn01; // LiftingPositionRound_2
	      R     "MAL1S033Par".Par.Switches1.StaOn00; // LiftingPositionRound_1
	      U     "MAL1S033Par".Par.Switches1.StaOn00; // LiftingPositionRound_1
	      SPB   Rnd1;
	      U     "MAL1S033Par".Par.Switches1.StaOn01; // LiftingPositionRound_2
	      SPB   Rnd2;
	      U     "MAL1S033Par".Par.Switches1.StaOn02; // LiftingPositionRound_3
	      SPB   Rnd3;
	      U     "MAL1S033Par".Par.Switches1.StaOn03; // LiftingPositionRound_4
	      SPB   Rnd4;
	      U     "MAL1S033Par".Par.Switches1.StaOn04; // LiftingPositionRound_5
	      SPB   Rnd5;
	      U     "MAL1S033Par".Par.Switches1.StaOn05; // LiftingPositionRound_6
	      SPB   Rnd6;
	      SPA   E700;
	Rnd1: NOP   0;
	      L     "MAL1S033Par".RecipeHeader.Loading.LoadingLevelRound_1;
	      T     "MAL1S033Par".Par.MachineValue.SOLLWERT_HUBZUG1_HOEHE;
	      T     "MAL1S033Par".Par.MachineValue.SOLLWERT_HUBZUG2_HOEHE;
	      L     "MAL1S033Par".RecipeHeader.Loading.LoadingSpeed_1;
	      T     "MAL1S033Par".Par.MachineValue.SollwertFahrantrieb;
	      SPA   E700;
	Rnd2: NOP   0;
	      L     "MAL1S033Par".RecipeHeader.Loading.LoadingLevelRound_2;
	      T     "MAL1S033Par".Par.MachineValue.SOLLWERT_HUBZUG1_HOEHE;
	      T     "MAL1S033Par".Par.MachineValue.SOLLWERT_HUBZUG2_HOEHE;
	      L     "MAL1S033Par".RecipeHeader.Loading.LoadingSpeed_2;
	      T     "MAL1S033Par".Par.MachineValue.SollwertFahrantrieb;
	      SPA   E700;
	Rnd3: NOP   0;
	      L     "MAL1S033Par".RecipeHeader.Loading.LoadingLevelRound_3;
	      T     "MAL1S033Par".Par.MachineValue.SOLLWERT_HUBZUG1_HOEHE;
	      T     "MAL1S033Par".Par.MachineValue.SOLLWERT_HUBZUG2_HOEHE;
	      L     "MAL1S033Par".RecipeHeader.Loading.LoadingSpeed_3;
	      T     "MAL1S033Par".Par.MachineValue.SollwertFahrantrieb;
	      SPA   E700;
	Rnd4: NOP   0;
	      L     "MAL1S033Par".Par.ParIntMachine.LoadingLevelRound_4;
	      T     "MAL1S033Par".Par.MachineValue.SOLLWERT_HUBZUG1_HOEHE;
	      T     "MAL1S033Par".Par.MachineValue.SOLLWERT_HUBZUG2_HOEHE;
	      L     "MAL1S033Par".RecipeHeader.Loading.LoadingSpeed_3;
	      T     "MAL1S033Par".Par.MachineValue.SollwertFahrantrieb;
	      SPA   E700;
	Rnd5: NOP   0;
	      L     "MAL1S033Par".Par.ParIntMachine.LoadingLevelRound_5;
	      T     "MAL1S033Par".Par.MachineValue.SOLLWERT_HUBZUG1_HOEHE;
	      T     "MAL1S033Par".Par.MachineValue.SOLLWERT_HUBZUG2_HOEHE;
	      L     "MAL1S033Par".RecipeHeader.Loading.LoadingSpeed_3;
	      T     "MAL1S033Par".Par.MachineValue.SollwertFahrantrieb;
	      SPA   E700;
	Rnd6: NOP   0;
	      L     "MAL1S033Par".Par.ParIntMachine.LoadingLevelRound_6;
	      T     "MAL1S033Par".Par.MachineValue.SOLLWERT_HUBZUG1_HOEHE;
	      T     "MAL1S033Par".Par.MachineValue.SOLLWERT_HUBZUG2_HOEHE;
	      L     "MAL1S033Par".RecipeHeader.Loading.LoadingSpeed_3;
	      T     "MAL1S033Par".Par.MachineValue.SollwertFahrantrieb;
	      SPA   E700;
	E700: NOP   0;
	NETWORK
	TITLE =Sub 7010: Kilning  loading finished
	      L     0;
	      L     "MAL1S033".ToSSW.InPrevSecDB;
	      ==I   ;
	      SPB   fin;
	      O(;
	      U     "MAL1S017Par".Par.FlagFunction_1.FinishUnloading;
	      U     "MAL1S033".PCWrite.ExtFuncOn.FinishLoading; // PIC command "finish loading"
	      O       "MAL1S017Par".Par.FlagFunction_1.StepCleaning;
	      U     "MAL1S017".PCRead.Step.StEmptied;
	      U(    ;
	      AUF   "MAL1S017";
	      L DBNO;
	      L     "MAL1S033".ToSSW.InPrevSecDB;
	      ==I;
	      )     ;
	      )     ;
	      O(;
	      U     "MAL1S018Par".Par.FlagFunction_1.FinishUnloading;
	      U     "MAL1S033".PCWrite.ExtFuncOn.FinishLoading; // PIC command "finish loading"
	      O       "MAL1S018Par".Par.FlagFunction_1.StepCleaning;
	      U     "MAL1S018".PCRead.Step.StEmptied;
	      U(    ;
	      AUF   "MAL1S018";
	      L DBNO;
	      L     "MAL1S033".ToSSW.InPrevSecDB;
	      ==I;
	      )     ;
	      )     ;
	      O(;
	      U     "MAL1S019Par".Par.FlagFunction_1.FinishUnloading;
	      U     "MAL1S033".PCWrite.ExtFuncOn.FinishLoading; // PIC command "finish loading"
	      O       "MAL1S019Par".Par.FlagFunction_1.StepCleaning;
	      U     "MAL1S019".PCRead.Step.StEmptied;
	      U(    ;
	      AUF   "MAL1S019";
	      L DBNO;
	      L     "MAL1S033".ToSSW.InPrevSecDB;
	      ==I;
	      )     ;
	      )     ;
	      O(;
	      U     "MAL1S020Par".Par.FlagFunction_1.FinishUnloading;
	      U     "MAL1S033".PCWrite.ExtFuncOn.FinishLoading; // PIC command "finish loading"
	      O       "MAL1S020Par".Par.FlagFunction_1.StepCleaning;
	      U     "MAL1S020".PCRead.Step.StEmptied;
	      U(    ;
	      AUF   "MAL1S020";
	      L DBNO;
	      L     "MAL1S033".ToSSW.InPrevSecDB;
	      ==I;
	      )     ;
	      )     ;
	      O(;
	      U     "MAL1S021Par".Par.FlagFunction_1.FinishUnloading;
	      U     "MAL1S033".PCWrite.ExtFuncOn.FinishLoading; // PIC command "finish loading"
	      O       "MAL1S021Par".Par.FlagFunction_1.StepCleaning;
	      U     "MAL1S021".PCRead.Step.StEmptied;
	      U(    ;
	      AUF   "MAL1S021";
	      L DBNO;
	      L     "MAL1S033".ToSSW.InPrevSecDB;
	      ==I;
	      )     ;
	      )     ;
	      O(;
	      U     "MAL1S022Par".Par.FlagFunction_1.FinishUnloading;
	      U     "MAL1S033".PCWrite.ExtFuncOn.FinishLoading; // PIC command "finish loading"
	      O       "MAL1S022Par".Par.FlagFunction_1.StepCleaning;
	      U     "MAL1S022".PCRead.Step.StEmptied;
	      U(    ;
	      AUF   "MAL1S022";
	      L DBNO;
	      L     "MAL1S033".ToSSW.InPrevSecDB;
	      ==I;
	      )     ;
	      )     ;
	      O(;
	      U     "MAL1S023Par".Par.FlagFunction_1.FinishUnloading;
	      U     "MAL1S033".PCWrite.ExtFuncOn.FinishLoading; // PIC command "finish loading"
	      O       "MAL1S023Par".Par.FlagFunction_1.StepCleaning;
	      U     "MAL1S023".PCRead.Step.StEmptied;
	      U(    ;
	      AUF   "MAL1S023";
	      L DBNO;
	      L     "MAL1S033".ToSSW.InPrevSecDB;
	      ==I;
	      )     ;
	      )     ;
	      O(;
	      U     "MAL1S024Par".Par.FlagFunction_1.FinishUnloading;
	      U     "MAL1S033".PCWrite.ExtFuncOn.FinishLoading; // PIC command "finish loading"
	      O       "MAL1S024Par".Par.FlagFunction_1.StepCleaning;
	      U     "MAL1S024".PCRead.Step.StEmptied;
	      U(    ;
	      AUF   "MAL1S024";
	      L DBNO;
	      L     "MAL1S033".ToSSW.InPrevSecDB;
	      ==I;
	      )     ;
	      )     ;
	      O(    ;
	      U     "MAL1S033Par".Par.FlagFunction_1.StepLoading; // Step loading
	      UN    "MAL1S033".ToASW.InfSameJobPrevSec;
	      U     "MAL1S033".PCWrite.ExtFuncOn.FinishLoading; // PIC command "finish loading"
	      )     ;
	      U     "MAL1S033".ToASW.InfDataReady;
	      U     "MAL1S033".PCRead.Step.StActive;
	      S     "MAL1S033Par".Par.FlagFunction_1.LoadEnd;
	//
	      U     "MAL1S033".PCWrite.ExtFuncOn.FinishLoading; // PIC command "finish loading"
	      R     "MAL1S033".PCWrite.ExtFuncOn.FinishLoading; // PIC command "finish loading"
	//
	      U     "MAL1S033Par".Par.FlagFunction_1.LoadEnd;
	      U     "MAL1S033Par".Par.FlagFunction_1.StepLoading; // Step loading
	      FP    "MAL1S033Par".Par.FlagFunction_0.ImpulsSollposition;
	      =     "MAL1S033Par".Par.FlagFunction_0.MerkerSollpositionFP;
	      U     "MAL1S033Par".Par.FlagFunction_0.MerkerSollpositionFP;
	      SPBN  fin;
	      L     G292M.A_3211_MXZ41MA.Ma.OutPositionAngle;
	      L     "MAL1S033Par".Par.ParIntProcess.LoadingOverlap;
	      +I    ;
	      T     G292M.A_3211_MXZ41MA.Ma.InPositionTarget;
	//???      SET
	//???      S     "G292M".TurningTo_Parkposition    // G292M.A_3211_MXZ41MA..Ma.InAdjusting
	// Beladehöhe speichern
	      L     "MAL1S033Par".Par.MachineValue.SOLLWERT_HUBZUG1_HOEHE;
	      T     "MAL1S033Par".Par.ParIntMachine.LastLoadingLevel; // saved loading value
	fin:  NOP   0;
	E701: NOP   0;
	NETWORK
	TITLE =Sub 7020: Step start process kilning
	      U     "MAL1S033".ToASW.InfDataReady;
	      U     "MAL1S033".PCRead.Step.StActive;
	//    U     "MAL1S033".PCWrite.ExtFuncOn.StartProcess    // PIC command "start process kilning"
	      U     "MAL1S033Par".Par.FlagFunction_1.LoadEnd;
	      U(    ;
	      O     G292M.A_3211_MXZ41MA.A_3211_BZS43.StTrue;    // sensor zero point


	      )     ;
	      S     "MAL1S033Par".Par.FlagFunction_1.FinishLoading; // start process kilning
	      R     "MAL1S033Par".Par.FlagFunction_1.LoadEnd;
	//
	      U     "MAL1S033".PCWrite.ExtFuncOn.StartProcess; // PIC command "start process kilning"
	      R     "MAL1S033".PCWrite.ExtFuncOn.StartProcess; // PIC command "start process kilning"
	//
	      U     "MAL1S033".ToASW.InfDataReady;
	      U(    ;
	      O     "MAL1S033".PCRead.Step.StActive;
	      O     "MAL1S033".PCRead.Step.StReady;
	      )     ;
	      U     "MAL1S033Par".Par.FlagProcess.ProcessActive;
	      U     G292M.A_3211_MXZ41MA.A_3211_BZS43.StTrue;    // sensor zero point
	      SPBN  E702;

	      L     50; //jk
	      +I    ;
	      T     "MAL1S033Par".Par.MachineValue.SOLLWERT_HUBZUG1_HOEHE;

	      L     50; //jk
	      +I    ;
	      T     "MAL1S033Par".Par.MachineValue.SOLLWERT_HUBZUG2_HOEHE;
	      L     3;

	E702: NOP   0;
	NETWORK
	NETWORK
	TITLE =ASW_9000: Step cleaning
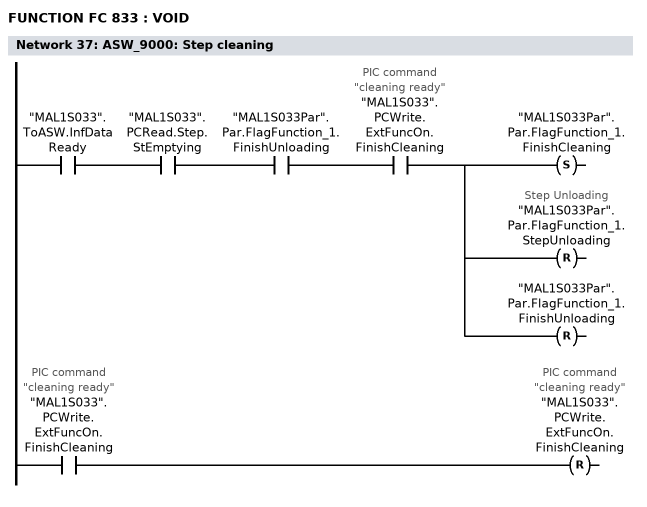
	      U     "MAL1S033".ToASW.InfDataReady;
	      U     "MAL1S033".PCRead.Step.StEmptying;
	      U     "MAL1S033Par".Par.FlagFunction_1.FinishUnloading;
	      U     "MAL1S033".PCWrite.ExtFuncOn.FinishCleaning; // PIC command "cleaning ready"
	      S     "MAL1S033Par".Par.FlagFunction_1.FinishCleaning;
	      R     "MAL1S033Par".Par.FlagFunction_1.StepUnloading; // Step Unloading
	      R     "MAL1S033Par".Par.FlagFunction_1.FinishUnloading;
	//
	      U     "MAL1S033".PCWrite.ExtFuncOn.FinishCleaning; // PIC command "cleaning ready"
	      R     "MAL1S033".PCWrite.ExtFuncOn.FinishCleaning; // PIC command "cleaning ready"
	NETWORK
	TITLE =ASW_9080: Send section date to PIC after germination

	      AUF   "MAL1S033";
	      U     "MAL1S033".PCRead.Step.StEmptying;
	      FP    "MAL1S033Par".Par.FlagProcess.FP_SendResultToPIC;
	      SPBN  E908;
	//

	E908: NOP   0;
	NETWORK
	TITLE =ASW_10000: ILO functions
	//
	      U     "MAL1S033".SecAc.Sta1On.Inf08;
	      =     "MAL1S033".Gr.All.Spare04;

	//- Little help for PIC-People
	      U     "MAL1S033".SecAc.Sta1On.Inf08;
	      SPB   RSM;
	      L     0;
	      T     "MAL1S033Par".Ilo.Code_ILO_Funktion0; // FCM 33 LINE 1 SEC 33 KILN 2
	RSM:  NOP   0;

	//  no ILO-mode >> cmd manual off to all used groups and reset all flags
	      U     "MAL1S033".SecAc.Sta1On.Inf08;
	      FN    "MAL1S033Par".Ilo.Flag.EdgeILOModeOn;
	      S     "MAL1S033Par".Ilo.GrCMDManOff[1]; // (ManOff)
	      R     "MAL1S033Par".Ilo.GrCMDManAdditional.Cmd1[1];
	      R     "MAL1S033Par".Ilo.GrCMDManAdditional.Cmd2[2];
	//  Gr-cmd manual OFF
	      S     "G291M".Gr.CmdManualOff; // LIFTING DEVICE KILN 2
	      S     "G292M".Gr.CmdManualOff; // TRAVELLING DRIVE KILN 2
	      S     "G293M".Gr.CmdManualOff; // UNLOADING / LOADING SCREW KILN 2
	      S     "G294M".Gr.CmdManualOff; // DISCHARGE DOOR KILN 2
	      S     "G297M".Gr.CmdManualOff; // FAN KILN 2
	      S     "G298M".Gr.CmdManualOff; // FRESH AIR LOUVER KILN 2
	      S     "G299M".Gr.CmdManualOff; // RECYCLING AIR FLAP KILN 2
	      S     "G302M".Gr.CmdManualOff; // HEATING KILN 2
	      S     "G303M".Gr.CmdManualOff; // LOUVER AIR HEATER KILN 2
	      S     "G304M".Gr.CmdManualOff; // WITHERING AIR KILN 2
	      S     "G305M".Gr.CmdManualOff; // CHAIN CONVEYOR 9002 KILN 2
	//  RESET ADDITIONAL CMD`S
	      R     "G291M".USW14; // ILO-cmd
	      R     "G291M".USW15; // ILO-cmd
	      R     "G292M".USW14; // ILO-cmd
	      R     "G292M".USW15; // ILO-cmd
	      R     "G293M".USW14; // ILO-cmd
	      R     "G293M".USW15; // ILO-cmd
	      R     "G294M".USW14; // ILO-cmd
	      R     "G294M".USW15; // ILO-cmd
	      R     "G297M".USW14; // ILO-cmd
	      R     "G297M".USW15; // ILO-cmd
	      R     "G298M".USW14; // ILO-cmd
	      R     "G298M".USW15; // ILO-cmd
	      R     "G299M".USW14; // ILO-cmd
	      R     "G299M".USW15; // ILO-cmd
	      R     "G302M".USW14; // ILO-cmd
	      R     "G302M".USW15; // ILO-cmd
	      R     "G303M".USW14; // ILO-cmd
	      R     "G303M".USW15; // ILO-cmd
	      R     "G304M".USW14; // ILO-cmd
	      R     "G304M".USW15; // ILO-cmd
	      R     "G305M".USW14; // ILO-cmd
	      R     "G305M".USW15; // ILO-cmd
	//
	      NOP   0;
	// --- FCM 01 - Lifting devices ---
	    L "MAL1S033Par".Ilo.ILOMode;
	    L  1;
	    <>I;
	    SPB IO1;
	// man on
	      U     "MAL1S033Par".Ilo.GrCMDManOn[1];
	      S     "G291M".Gr.InManual; // LIFTING DEVICE KILN 2
	      R     "MAL1S033Par".Ilo.GrCMDManOn[1];
	// man off
	      U     "MAL1S033Par".Ilo.GrCMDManOff[1];
	      S     "G291M".Gr.CmdManualOff; // LIFTING DEVICE KILN 2
	      R     "G291M".Gr.InManual; // LIFTING DEVICE KILN 2
	      R     "G291M".USW14; // ILO-cmd
	      R     "G291M".USW15; // ILO-cmd
	      R     "MAL1S033Par".Ilo.GrCMDManOff[1];
	      R     "MAL1S033Par".Ilo.GrCMDManAdditional.Cmd1[1];
	      R     "MAL1S033Par".Ilo.GrCMDManAdditional.Cmd2[1];
	// man start
	      U     "MAL1S033Par".Ilo.GrCMDManStart[1];
	      S     "G291M".Gr.CmdOn; // LIFTING DEVICE KILN 2
	      S     "G291M".Gr.CmdContinue; // LIFTING DEVICE KILN 2
	      R     "MAL1S033Par".Ilo.GrCMDManStart[1];
	      U     "MAL1S033Par".Ilo.GrCMDManStart[2];
	      R     "MAL1S033Par".Ilo.GrCMDManStart[2];
	// man stop
	      U     "MAL1S033Par".Ilo.GrCMDManStop[1];
	      S     "G291M".Gr.CmdOff; // LIFTING DEVICE KILN 2
	      R     "MAL1S033Par".Ilo.GrCMDManStop[1];
	// man fault reset
	      U     "MAL1S033Par".Ilo.GrCMDManFaultReset[1];
	      S     "G291M".Gr.CmdFaultReset; // LIFTING DEVICE KILN 2
	      R     "MAL1S033Par".Ilo.GrCMDManFaultReset[1];
	// moving direction
	      UN    "G291M".Gr.InManual; // LIFTING DEVICE KILN 2
	      O(    ;
	      L     "MAL1S033Par".Ilo.Code_ILO_Funktion0;
	      L     100;
	      <>I   ;
	      )     ;
	      SPB   Stat;
	      UN    "MAL1S033Par".Ilo.GrCMDManAdditional.Cmd1[1];
	      UN    "MAL1S033Par".Ilo.GrCMDManAdditional.Cmd2[1];
	      L     "MAL1S033Par".Par.MachineValue.SOLLWERT_HUBZUG1_HOEHE;
	      SPB   Tpos;
	      U     "MAL1S033Par".Ilo.GrCMDManAdditional.Cmd1[1]; // ManUp
	      L     2000; // 1850mm + Offset = 2000mm
	      SPB   Tpos;
	      U     "MAL1S033Par".Ilo.GrCMDManAdditional.Cmd2[1]; // ManDown
	      L     0; // 0mm
	      SPB   Tpos;
	      SPA   Stat;
	// target position
	Tpos: NOP   0;
	      T     "MAL1S033Par".Par.ParIntProcess.TarPos_ILO_LiftDev;
	Stat: NOP   0;
	IO1 : NOP   0;
	      NOP   0;
	// --- FCM 04 - Fans ---
	    L "MAL1S033Par".Ilo.ILOMode;
	    L  4;
	    <>I;
	    SPB IO4;
	// man on
	      U     "MAL1S033Par".Ilo.GrCMDManOn[1];
	      S     "G297M".Gr.InManual; // FAN KILN 2
	      R     "MAL1S033Par".Ilo.GrCMDManOn[1];
	// man off
	      U     "MAL1S033Par".Ilo.GrCMDManOff[1];
	      S     "G297M".Gr.CmdManualOff; // FAN KILN 2
	      R     "G297M".Gr.InManual; // FAN KILN 2
	      R     "G297M".USW14; // ILO-cmd
	      R     "G297M".USW15; // ILO-cmd
	      R     "MAL1S033Par".Ilo.GrCMDManOff[1];
	      R     "MAL1S033Par".Ilo.GrCMDManAdditional.Cmd1[1];
	      R     "MAL1S033Par".Ilo.GrCMDManAdditional.Cmd2[1];
	// man start
	      U     "MAL1S033Par".Ilo.GrCMDManStart[1];
	      S     "G297M".Gr.CmdOn; // FAN KILN 2
	      S     "G297M".Gr.CmdContinue; // FAN KILN 2
	      R     "MAL1S033Par".Ilo.GrCMDManStart[1];
	      U     "MAL1S033Par".Ilo.GrCMDManStart[2];
	      R     "MAL1S033Par".Ilo.GrCMDManStart[2];
	// man stop
	      U     "MAL1S033Par".Ilo.GrCMDManStop[1];
	      S     "G297M".Gr.CmdOff; // FAN KILN 2
	      R     "MAL1S033Par".Ilo.GrCMDManStop[1];
	// man fault reset
	      U     "MAL1S033Par".Ilo.GrCMDManFaultReset[1];
	      S     "G297M".Gr.CmdFaultReset; // FAN KILN 2
	      R     "MAL1S033Par".Ilo.GrCMDManFaultReset[1];
	// target position
	      UN    "G297M".Gr.InManual; // FAN KILN 2
	      O(;
	      L     "MAL1S033Par".Ilo.Code_ILO_Funktion0;
	      L     400;
	      <>I;
	      );
	      SPB   F04a;
	      L     "MAL1S033Par".Ilo.SetpointInt01[1];
	      T     "MAL1S033Par".Par.ParIntProcess.Speed_ILO_Fan;
	F04a:  NOP   0;

	IO4 : NOP   0;
	      NOP   0;
	// --- FCM 05 - Fans with target air temperature ---
	    L "MAL1S033Par".Ilo.ILOMode;
	    L  5;
	    <>I;
	    SPB IO5;
	// man on
	      U     "MAL1S033Par".Ilo.GrCMDManOn[1];
	      S     "G297M".Gr.InManual; // FAN KILN 2
	      S     "G299M".Gr.InManual; // RECYCLING AIR FLAP KILN 2
	      S     "G299M".Gr.CmdOn; // No Button: RECYCLING AIR FLAP KILN 2
	      S     "G299M".Gr.CmdContinue; // No Button RECYCLING AIR FLAP KILN 2
	      S     "G302M".Gr.InManual; // HEATING KILN 2
	      S     "G302M".Gr.CmdOn; // No Button: HEATING KILN 2
	      S     "G302M".Gr.CmdContinue; // No Button HEATING KILN 2
	      S     "G303M".Gr.InManual; // LOUVER AIR HEATER KILN 2
	      S     "G303M".Gr.CmdOn; // No Button: LOUVER AIR HEATER KILN 2
	      S     "G303M".Gr.CmdContinue; // No Button LOUVER AIR HEATER KILN 2
	      S     "G298M".Gr.InManual; // FRESH AIR LOUVER KILN 2
	      S     "G298M".Gr.CmdOn; // No Button: FRESH AIR LOUVER KILN 2
	      S     "G298M".Gr.CmdContinue; // No Button FRESH AIR LOUVER KILN 2
	      S     "G304M".Gr.InManual; // WITHERING AIR KILN 2
	      S     "G304M".Gr.CmdOn; // No Button: WITHERING AIR KILN 2
	      S     "G304M".Gr.CmdContinue; // No Button WITHERING AIR KILN 2
	      R     "MAL1S033Par".Ilo.GrCMDManOn[1];
	// man off
	      U     "MAL1S033Par".Ilo.GrCMDManOff[1];
	      S     "G297M".Gr.CmdManualOff; // FAN KILN 2
	      R     "G297M".Gr.InManual; // FAN KILN 2
	      R     "G297M".USW14; // ILO-cmd
	      R     "G297M".USW15; // ILO-cmd
	      S     "G299M".Gr.CmdManualOff; // RECYCLING AIR FLAP KILN 2
	      R     "G299M".Gr.InManual; // RECYCLING AIR FLAP KILN 2
	      R     "G299M".USW14; // ILO-cmd
	      R     "G299M".USW15; // ILO-cmd
	      S     "G302M".Gr.CmdManualOff; // HEATING KILN 2
	      R     "G302M".Gr.InManual; // HEATING KILN 2
	      R     "G302M".USW14; // ILO-cmd
	      R     "G302M".USW15; // ILO-cmd
	      S     "G303M".Gr.CmdManualOff; // LOUVER AIR HEATER KILN 2
	      R     "G303M".Gr.InManual; // LOUVER AIR HEATER KILN 2
	      R     "G303M".USW14; // ILO-cmd
	      R     "G303M".USW15; // ILO-cmd
	      S     "G298M".Gr.CmdManualOff; // FRESH AIR LOUVER KILN 2
	      R     "G298M".Gr.InManual; // FRESH AIR LOUVER KILN 2
	      R     "G298M".USW14; // ILO-cmd
	      R     "G298M".USW15; // ILO-cmd
	      S     "G304M".Gr.CmdManualOff; // WITHERING AIR KILN 2
	      R     "G304M".Gr.InManual; // WITHERING AIR KILN 2
	      R     "G304M".USW14; // ILO-cmd
	      R     "G304M".USW15; // ILO-cmd
	      R     "MAL1S033Par".Ilo.GrCMDManOff[1];
	      R     "MAL1S033Par".Ilo.GrCMDManAdditional.Cmd1[1];
	      R     "MAL1S033Par".Ilo.GrCMDManAdditional.Cmd2[1];
	// man start
	      U     "MAL1S033Par".Ilo.GrCMDManStart[1];
	      S     "G297M".Gr.CmdOn; // FAN KILN 2
	      S     "G297M".Gr.CmdContinue; // FAN KILN 2
	      S     "G299M".Gr.CmdOn; // RECYCLING AIR FLAP KILN 2
	      S     "G299M".Gr.CmdContinue; // RECYCLING AIR FLAP KILN 2
	      S     "G302M".Gr.CmdOn; // HEATING KILN 2
	      S     "G302M".Gr.CmdContinue; // HEATING KILN 2
	      S     "G303M".Gr.CmdOn; // LOUVER AIR HEATER KILN 2
	      S     "G303M".Gr.CmdContinue; // LOUVER AIR HEATER KILN 2
	      S     "G298M".Gr.CmdOn; // FRESH AIR LOUVER KILN 2
	      S     "G298M".Gr.CmdContinue; // FRESH AIR LOUVER KILN 2
	      S     "G304M".Gr.CmdOn; // WITHERING AIR KILN 2
	      S     "G304M".Gr.CmdContinue; // WITHERING AIR KILN 2
	      R     "MAL1S033Par".Ilo.GrCMDManStart[1];
	      U     "MAL1S033Par".Ilo.GrCMDManStart[2];
	      R     "MAL1S033Par".Ilo.GrCMDManStart[2];
	// man stop
	      U     "MAL1S033Par".Ilo.GrCMDManStop[1];
	      S     "G297M".Gr.CmdOff; // FAN KILN 2
	      S     "G299M".Gr.CmdOff; // RECYCLING AIR FLAP KILN 2
	      S     "G302M".Gr.CmdOff; // HEATING KILN 2
	      S     "G303M".Gr.CmdOff; // LOUVER AIR HEATER KILN 2
	      S     "G298M".Gr.CmdOff; // FRESH AIR LOUVER KILN 2
	      S     "G304M".Gr.CmdOff; // WITHERING AIR KILN 2
	      R     "MAL1S033Par".Ilo.GrCMDManStop[1];
	// man fault reset
	      U     "MAL1S033Par".Ilo.GrCMDManFaultReset[1];
	      S     "G297M".Gr.CmdFaultReset; // FAN KILN 2
	      S     "G299M".Gr.CmdFaultReset; // RECYCLING AIR FLAP KILN 2
	      S     "G302M".Gr.CmdFaultReset; // HEATING KILN 2
	      S     "G303M".Gr.CmdFaultReset; // LOUVER AIR HEATER KILN 2
	      S     "G298M".Gr.CmdFaultReset; // FRESH AIR LOUVER KILN 2
	      S     "G304M".Gr.CmdFaultReset; // WITHERING AIR KILN 2
	      R     "MAL1S033Par".Ilo.GrCMDManFaultReset[1];
	// target position
	      UN    "G297M".Gr.InManual; // FAN KILN 2
	      O(;
	      L     "MAL1S033Par".Ilo.Code_ILO_Funktion0;
	      L     500;
	      <>I;
	      );
	      SPB   F05b;
	      L     "MAL1S033Par".Ilo.SetpointInt01[1];
	      T     "MAL1S033Par".Par.ParIntProcess.Speed_ILO_Fan;
	F05b:  NOP   0;
	IO5 : NOP   0;
	      NOP   0;
	// --- FCM 06 - Fresh air flap ---
	    L "MAL1S033Par".Ilo.ILOMode;
	    L  6;
	    <>I;
	    SPB IO6;
	// man on
	      U     "MAL1S033Par".Ilo.GrCMDManOn[1];
	      S     "G298M".Gr.InManual; // FRESH AIR LOUVER KILN 2
	      R     "MAL1S033Par".Ilo.GrCMDManOn[1];
	// man off
	      U     "MAL1S033Par".Ilo.GrCMDManOff[1];
	      S     "G298M".Gr.CmdManualOff; // FRESH AIR LOUVER KILN 2
	      R     "G298M".Gr.InManual; // FRESH AIR LOUVER KILN 2
	      R     "G298M".USW14; // ILO-cmd
	      R     "G298M".USW15; // ILO-cmd
	      R     "MAL1S033Par".Ilo.GrCMDManOff[1];
	      R     "MAL1S033Par".Ilo.GrCMDManAdditional.Cmd1[1];
	      R     "MAL1S033Par".Ilo.GrCMDManAdditional.Cmd2[1];
	// man start
	      U     "MAL1S033Par".Ilo.GrCMDManStart[1];
	      S     "G298M".Gr.CmdOn; // FRESH AIR LOUVER KILN 2
	      S     "G298M".Gr.CmdContinue; // FRESH AIR LOUVER KILN 2
	      R     "MAL1S033Par".Ilo.GrCMDManStart[1];
	      U     "MAL1S033Par".Ilo.GrCMDManStart[2];
	      R     "MAL1S033Par".Ilo.GrCMDManStart[2];
	// man stop
	      U     "MAL1S033Par".Ilo.GrCMDManStop[1];
	      S     "G298M".Gr.CmdOff; // FRESH AIR LOUVER KILN 2
	      R     "MAL1S033Par".Ilo.GrCMDManStop[1];
	// man fault reset
	      U     "MAL1S033Par".Ilo.GrCMDManFaultReset[1];
	      S     "G298M".Gr.CmdFaultReset; // FRESH AIR LOUVER KILN 2
	      R     "MAL1S033Par".Ilo.GrCMDManFaultReset[1];
	// moving direction
	//
	// target position
	      UN    "G298M".Gr.InManual; // FRESH AIR LOUVER KILN 2
	      SPB   F06b;
	      L     "MAL1S033Par".Ilo.SetpointInt01[1];
	      T     "MAL1S033Par".Par.ParIntProcess.TarPos_ILO_FreshAir;
	F06b:  NOP   0;

	IO6 : NOP   0;
	      NOP   0;
	// --- FCM 07 - Recycling air flap ---
	    L "MAL1S033Par".Ilo.ILOMode;
	    L  7;
	    <>I;
	    SPB IO7;
	// man on
	      U     "MAL1S033Par".Ilo.GrCMDManOn[1];
	      S     "G299M".Gr.InManual; // RECYCLING AIR FLAP KILN 2
	      S     "G304M".Gr.InManual; // WITHERING AIR KILN 2
	      R     "MAL1S033Par".Ilo.GrCMDManOn[1];
	// man off
	      U     "MAL1S033Par".Ilo.GrCMDManOff[1];
	      S     "G299M".Gr.CmdManualOff; // RECYCLING AIR FLAP KILN 2
	      R     "G299M".Gr.InManual; // RECYCLING AIR FLAP KILN 2
	      R     "G299M".USW14; // ILO-cmd
	      R     "G299M".USW15; // ILO-cmd
	      S     "G304M".Gr.CmdManualOff; // WITHERING AIR KILN 2
	      R     "G304M".Gr.InManual; // WITHERING AIR KILN 2
	      R     "G304M".USW14; // ILO-cmd
	      R     "G304M".USW15; // ILO-cmd
	      R     "MAL1S033Par".Ilo.GrCMDManOff[1];
	      R     "MAL1S033Par".Ilo.GrCMDManAdditional.Cmd1[1];
	      R     "MAL1S033Par".Ilo.GrCMDManAdditional.Cmd2[1];
	// man start
	      U     "MAL1S033Par".Ilo.GrCMDManStart[1];
	      S     "G299M".Gr.CmdOn; // RECYCLING AIR FLAP KILN 2
	      S     "G299M".Gr.CmdContinue; // RECYCLING AIR FLAP KILN 2
	      S     "G304M".Gr.CmdOn; // WITHERING AIR KILN 2
	      S     "G304M".Gr.CmdContinue; // WITHERING AIR KILN 2
	      R     "MAL1S033Par".Ilo.GrCMDManStart[1];
	      U     "MAL1S033Par".Ilo.GrCMDManStart[2];
	      R     "MAL1S033Par".Ilo.GrCMDManStart[2];
	// man stop
	      U     "MAL1S033Par".Ilo.GrCMDManStop[1];
	      S     "G299M".Gr.CmdOff; // RECYCLING AIR FLAP KILN 2
	      S     "G304M".Gr.CmdOff; // WITHERING AIR KILN 2
	      R     "MAL1S033Par".Ilo.GrCMDManStop[1];
	// man fault reset
	      U     "MAL1S033Par".Ilo.GrCMDManFaultReset[1];
	      S     "G299M".Gr.CmdFaultReset; // RECYCLING AIR FLAP KILN 2
	      S     "G304M".Gr.CmdFaultReset; // WITHERING AIR KILN 2
	      R     "MAL1S033Par".Ilo.GrCMDManFaultReset[1];
	// moving direction
	//
	// target position
	      UN    "G299M".Gr.InManual; // RECYCLING AIR FLAP KILN 2
	      SPB   F07a;
	      L     "MAL1S033Par".Ilo.SetpointInt01[1];
	      T     "MAL1S033Par".Par.ParIntProcess.TarPos_ILO_RecycAir;
	F07a:  NOP   0;
	IO7 : NOP   0;
	      NOP   0;
	// --- FCM 09 - Floor drives ---
	    L "MAL1S033Par".Ilo.ILOMode;
	    L  9;
	    <>I;
	    SPB IO9;
	// man on
	      U     "MAL1S033Par".Ilo.GrCMDManOn[1];
	      S     "G292M".Gr.InManual; // TRAVELLING DRIVE KILN 2
	      R     "MAL1S033Par".Ilo.GrCMDManOn[1];
	// man off
	      U     "MAL1S033Par".Ilo.GrCMDManOff[1];
	      S     "G292M".Gr.CmdManualOff; // TRAVELLING DRIVE KILN 2
	      R     "G292M".Gr.InManual; // TRAVELLING DRIVE KILN 2
	      R     "G292M".USW14; // ILO-cmd
	      R     "G292M".USW15; // ILO-cmd
	      R     "MAL1S033Par".Ilo.GrCMDManOff[1];
	      R     "MAL1S033Par".Ilo.GrCMDManAdditional.Cmd1[1];
	      R     "MAL1S033Par".Ilo.GrCMDManAdditional.Cmd2[1];
	// man start
	      U     "MAL1S033Par".Ilo.GrCMDManStart[1];
	      S     "G292M".Gr.CmdOn; // TRAVELLING DRIVE KILN 2
	      S     "G292M".Gr.CmdContinue; // TRAVELLING DRIVE KILN 2
	      R     "MAL1S033Par".Ilo.GrCMDManStart[1];
	      U     "MAL1S033Par".Ilo.GrCMDManStart[2];
	      R     "MAL1S033Par".Ilo.GrCMDManStart[2];
	// man stop
	      U     "MAL1S033Par".Ilo.GrCMDManStop[1];
	      S     "G292M".Gr.CmdOff; // TRAVELLING DRIVE KILN 2
	      R     "MAL1S033Par".Ilo.GrCMDManStop[1];
	// man fault reset
	      U     "MAL1S033Par".Ilo.GrCMDManFaultReset[1];
	      S     "G292M".Gr.CmdFaultReset; // TRAVELLING DRIVE KILN 2
	      R     "MAL1S033Par".Ilo.GrCMDManFaultReset[1];
	f091: NOP   0;
	      UN    "G292M".Gr.InManual; // TRAVELLING DRIVE KILN 2
	      O     ;
	      UN    "MAL1S033Par".Ilo.GrCMDManAdditional.Cmd1[1];
	      UN    "MAL1S033Par".Ilo.GrCMDManAdditional.Cmd2[1];
	      SPB   f092;
	      U     "MAL1S033Par".Ilo.GrCMDManAdditional.Cmd1[1];
	      =     "G292M".USW14; // ILO-cmd run fwd
	      U     "MAL1S033Par".Ilo.GrCMDManAdditional.Cmd2[1];
	      =     "G292M".USW15; // ILO-cmd run rev
	// target position
	      L     "MAL1S033Par".Ilo.SetpointInt01[1];
	      T     "MAL1S033Par".Par.ParIntProcess.Speed_ILO_FloorRotating;
	f092: NOP   0;

	IO9 : NOP   0;
	      NOP   0;
	// --- FCM 10 - Floor drives and lifting devices ---
	    L "MAL1S033Par".Ilo.ILOMode;
	    L  10;
	    <>I;
	    SPB IO10;
	// man on
	      U     "MAL1S033Par".Ilo.GrCMDManOn[1];
	      S     "G291M".Gr.InManual; // LIFTING DEVICE KILN 2
	      S     "G291M".Gr.CmdOn; // No Button: LIFTING DEVICE KILN 2
	      S     "G291M".Gr.CmdContinue; // No Button LIFTING DEVICE KILN 2
	      S     "G292M".Gr.InManual; // TRAVELLING DRIVE KILN 2
	      R     "MAL1S033Par".Ilo.GrCMDManOn[1];
	// man off
	      U     "MAL1S033Par".Ilo.GrCMDManOff[1];
	      S     "G291M".Gr.CmdManualOff; // LIFTING DEVICE KILN 2
	      R     "G291M".Gr.InManual; // LIFTING DEVICE KILN 2
	      R     "G291M".USW14; // ILO-cmd
	      R     "G291M".USW15; // ILO-cmd
	      S     "G292M".Gr.CmdManualOff; // TRAVELLING DRIVE KILN 2
	      R     "G292M".Gr.InManual; // TRAVELLING DRIVE KILN 2
	      R     "G292M".USW14; // ILO-cmd
	      R     "G292M".USW15; // ILO-cmd
	      R     "MAL1S033Par".Ilo.GrCMDManOff[1];
	      R     "MAL1S033Par".Ilo.GrCMDManAdditional.Cmd1[1];
	      R     "MAL1S033Par".Ilo.GrCMDManAdditional.Cmd2[1];
	// man start
	      U     "MAL1S033Par".Ilo.GrCMDManStart[1];
	      S     "G292M".Gr.CmdOn; // TRAVELLING DRIVE KILN 2
	      S     "G292M".Gr.CmdContinue; // TRAVELLING DRIVE KILN 2
	      R     "MAL1S033Par".Ilo.GrCMDManStart[1];
	      U     "MAL1S033Par".Ilo.GrCMDManStart[2];
	      S     "G291M".Gr.CmdOn; // LIFTING DEVICE KILN 2
	      S     "G291M".Gr.CmdContinue; // LIFTING DEVICE KILN 2
	      R     "MAL1S033Par".Ilo.GrCMDManStart[2];
	      U     "MAL1S033Par".Ilo.GrCMDManStart[3];
	      R     "MAL1S033Par".Ilo.GrCMDManStart[3];
	// man stop
	      U     "MAL1S033Par".Ilo.GrCMDManStop[1];
	      S     "G291M".Gr.CmdOff; // LIFTING DEVICE KILN 2
	      S     "G292M".Gr.CmdOff; // TRAVELLING DRIVE KILN 2
	      R     "MAL1S033Par".Ilo.GrCMDManStop[1];
	// man fault reset
	      U     "MAL1S033Par".Ilo.GrCMDManFaultReset[1];
	      S     "G291M".Gr.CmdFaultReset; // LIFTING DEVICE KILN 2
	      S     "G292M".Gr.CmdFaultReset; // TRAVELLING DRIVE KILN 2
	      R     "MAL1S033Par".Ilo.GrCMDManFaultReset[1];
	// moving direction
	f101: NOP   0;
	      UN    "G292M".Gr.InManual; // TRAVELLING DRIVE KILN 2
	      O     ;
	      UN    "MAL1S033Par".Ilo.GrCMDManAdditional.Cmd1[1];
	      UN    "MAL1S033Par".Ilo.GrCMDManAdditional.Cmd2[1];
	      SPB   f102;
	      U     "MAL1S033Par".Ilo.GrCMDManAdditional.Cmd1[1];
	      =     "G292M".USW14; // ILO-cmd run fwd
	      U     "MAL1S033Par".Ilo.GrCMDManAdditional.Cmd2[1];
	      =     "G292M".USW15; // ILO-cmd run rev
	// target speed floor drives
	      L     "MAL1S033Par".Ilo.SetpointInt01[1];
	      T     "MAL1S033Par".Par.ParIntProcess.Speed_ILO_FloorRotating;
	f102: NOP   0;
	      UN    "G291M".Gr.InManual; // LIFTING DEVICE KILN 2
	      O(    ;
	      L     "MAL1S033Par".Ilo.Code_ILO_Funktion0;
	      L     1000;
	      <>I   ;
	      )     ;
	      SPB   f103;
	// target position lifting devices
	      L     "MAL1S033Par".Ilo.SetpointInt02[1];
	      T     "MAL1S033Par".Par.ParIntProcess.TarPos_ILO_LiftDev;
	f103: NOP   0;

